(* Logix 5000 project; controller Ceca_1650T_Press 5069-L306ERM rev 32.11; software revision 32.02 *)

TASK MainTask (continuous, watchdog 500 ms) : MainProgram

MODULES
   Local : 5069-L306ERM (5069 0, rev 32.11)
END_MODULES

TYPE Recipe_Setup :
STRUCT
   AUTO_UPPER_ASSIST_POSITION : REAL;
   AUTO_UPPER_LIMIT_POSITION : REAL;
   R_DIECUSHION_AUTO_UP_ASSIST_POSITION : REAL;
   L_DIECUSHION_AUTO_UP_ASSIST_POSITION : REAL;
   L_DIECUSHION_AUTO_UP_LIMIT_POSITION : REAL;
   R_DIECUSHION_AUTO_UP_LIMIT_POSITION : REAL;
   SLIDE_SLOW_DOWN_SIGNAL_POSITION : REAL;
END_STRUCT
END_TYPE

TYPE SICK_AFX60_WS_DATA :   // Data structure for AFS60 / AFM60 WebServer
STRUCT
   Acceleration_Format : INT;
   Acceleration_HighLimit : DINT;
   Acceleration_LowLimit : DINT;
   CMR : DINT;
   CNR_D : DINT;
   CNR_N : DINT;
   CPR : DINT;
   CS : SINT;
   ESF : SINT;
   DirectionChange_Limit : DINT;
   MotionTime_Limit_seconds : DINT;
   PowerTime_Limit_seconds : DINT;
   StartsCCW_Limit : DINT;
   StartsCW_Limit : DINT;
   Position_HighLimit : DINT;
   Position_LowLimit : DINT;
   PresetValue : DINT;
   Scaling : SINT;
   SlaveSignOfLife : DINT;
   Temperature_Format : INT;
   Velocity_Format : INT;
   Velocity_HighLimit : DINT;
   Velocity_LowLimit : DINT;
   xErrorCode : DINT;
   xMsgRecordArray : SINT[4];
   SerialNo : DINT;
END_STRUCT
END_TYPE

ADD_ON_INSTRUCTION SICK_AFX60_A101WS_A103WS_AOI   (* revision 1.0, vendor SICK AG *)
VAR_IN_OUT
   InputAssembly_101WS_103WS : DINT[1]; {required}
   msgGetData : MESSAGE; {required}
   msgSetData : MESSAGE; {required}
   GetData : SICK_AFX60_WS_DATA; {required}
   SetData : SICK_AFX60_WS_DATA; {required}
END_VAR
VAR_INPUT
   ManualGetData : BOOL; {access Read Only}
END_VAR
VAR
   SizeInput : DINT; {access None}
   fbTON : FBD_TIMER; {access None}
   SickAFx_RESET_FaultHeader_Value : SINT; {access None}
   SET_ALL_in_Progress : SINT; {access None}
   Local_ManualGetData : SINT; {access None}
   AttributeList : DINT[24]; {access None}
   Count_Attributes : DINT; {access None}
   ACC_FORMAT : DINT; {access None}
   ACC_HIGH_LIMIT : DINT; {access None}
   ACC_LOW_LIMIT : DINT; {access None}
   CMR : DINT; {access None}
   CNR_D : DINT; {access None}
   CNR_N : DINT; {access None}
   CPR : DINT; {access None}
   CS : DINT; {access None}
   ESF : DINT; {access None}
   MAX_DIR_CHANGE : DINT; {access None}
   MAX_MOTION_TIME : DINT; {access None}
   MAX_POWER_TIME : DINT; {access None}
   MAX_STARTS_CCW : DINT; {access None}
   MAX_STARTS_CW : DINT; {access None}
   POS_HIGH_LIMIT : DINT; {access None}
   POS_LOW_LIMIT : DINT; {access None}
   PRESET_VALUE : DINT; {access None}
   SCALING : DINT; {access None}
   SLAVE_SIGN_OF_LIFE : DINT; {access None}
   TEMP_FORMAT : DINT; {access None}
   VELO_FORMAT : DINT; {access None}
   VELO_HIGH_LIMIT : DINT; {access None}
   VELO_LOW_LIMIT : DINT; {access None}
   arrReadData : DINT[10]; {access None}
   iAttribute : DINT;
   iStep : DINT;
   MAX_ATTRIBUTE : DINT; {access None}
   MIN_ATTRIBUTE : DINT; {access None}
   SERIAL_NO : DINT; {access Read Only}
   goto_iStep : DINT; {access None}
END_VAR

ROUTINE Logic   (* structured text *)
   (*=================================================================================
   Name:	AFX60 WebServer AOI
   Author:	SICK STEGMANN GMBH
   -----------------------------------------------------------------------------------
   Description:
   The routine supports the explicit data messaging between the Rockwell PLC and the
   SICK AFx60 encoder via EtherNet/IP. This routine makes it possible to equalize
   (read and write) a defined set of configuration parameters via EtherNet/IP.
   
   Version history:
   Date        | Version  | created under Logix V. | Author     | Remark
   -----------------------------------------------------------------------------------
   2015.05.21  | 1.0.0    | V21.00.00 CPR 9 SR 5.1 | SICK STD RP| Release version
   2015.06.03  | 1.0.1    | V21.00.00 CPR 9 SR 5.1 | SICK STD RP| AutoSave on Encoder change
   2015.07.06  | 1.0.2    | V21.00.00 CPR 9 SR 5.1 | SICK STD RP| Changed Param Update order
   ==================================================================================*)
   
   (*================================ GENERAL =======================================*)
   (*Initialize variables *)
   	MIN_ATTRIBUTE	:= 0;
   
   	SERIAL_NO      :=  MIN_ATTRIBUTE;
   	ESF            :=  1;
   	SCALING        :=  2;
   	ACC_FORMAT     :=  3;
   	ACC_HIGH_LIMIT :=  4;
   	ACC_LOW_LIMIT  :=  5;
   	CNR_D          :=  6;
   	CNR_N          :=  7;
   	CPR            :=  8;
   	CMR            :=  9;
   	CS             := 10;
   	MAX_DIR_CHANGE := 11;
   	MAX_MOTION_TIME:= 12;
   	MAX_POWER_TIME := 13;
   	MAX_STARTS_CCW := 14;
   	MAX_STARTS_CW  := 15;
   	POS_HIGH_LIMIT := 16;
   	POS_LOW_LIMIT  := 17;
   	PRESET_VALUE   := 18;
   	SLAVE_SIGN_OF_LIFE := 19;
   	TEMP_FORMAT        := 20;
   	VELO_FORMAT        := 21;
   	VELO_HIGH_LIMIT    := 22;
   	VELO_LOW_LIMIT     := 23;
   
   	MAX_ATTRIBUTE 		:= VELO_LOW_LIMIT;
   	Count_Attributes     := MAX_ATTRIBUTE + 1;
   
   	AttributeList[SERIAL_NO      ] :=   6; (* Attrib.ID of SerialNumber - Identity Object *)
   	AttributeList[ACC_FORMAT     ] :=  30; (* Attrib.ID of AccFormat *)
   	AttributeList[ACC_HIGH_LIMIT ] :=  33; (* Attrib.ID of AccHighLimit *)
   	AttributeList[ACC_LOW_LIMIT  ] :=  32; (* Attrib.ID of AccLowLimit *)
   	AttributeList[CMR            ] :=  17; (* Attrib.ID of CMR *)
   	AttributeList[CNR_D          ] := 127; (* Attrib.ID of CNR_D *)
   	AttributeList[CNR_N          ] := 126; (* Attrib.ID of CNR_N *)
   	AttributeList[CPR            ] :=  16; (* Attrib.ID of CPR *)
   	AttributeList[CS             ] :=  12; (* Attrib.ID of CS *)
   	AttributeList[ESF            ] := 125; (* Attrib.ID of ESF *)
   	AttributeList[MAX_DIR_CHANGE ] := 136; (* Attrib.ID of MaxDirChange *)
   	AttributeList[MAX_MOTION_TIME] := 134; (* Attrib.ID of MaxMotionTime *)
   	AttributeList[MAX_POWER_TIME ] := 135; (* Attrib.ID of MaxPowerTime *)
   	AttributeList[MAX_STARTS_CCW ] := 138; (* Attrib.ID of MaxStartsCCW *)
   	AttributeList[MAX_STARTS_CW  ] := 137; (* Attrib.ID of MaxStartsCW *)
   	AttributeList[POS_HIGH_LIMIT ] :=  23; (* Attrib.ID of PosHighLimit *)
   	AttributeList[POS_LOW_LIMIT  ] :=  22; (* Attrib.ID of PosLowLimit *)
   	AttributeList[PRESET_VALUE   ] :=  19; (* Attrib.ID of PresetValue *)
   	AttributeList[SCALING        ] :=  14; (* Attrib.ID of Scaling *)
   	AttributeList[SLAVE_SIGN_OF_LIFE] := 106; (* Attrib.ID of SlaveSignOfLife *)
   	AttributeList[TEMP_FORMAT       ] := 101; (* Attrib.ID of TempFormat *)
   	AttributeList[VELO_FORMAT       ] :=  25; (* Attrib.ID of VeloFormat *)
   	AttributeList[VELO_HIGH_LIMIT   ] :=  28; (* Attrib.ID of VeloHighLimit *)
   	AttributeList[VELO_LOW_LIMIT    ] :=  27; (* Attrib.ID of VeloLowLimit *)
   (* END INIT *)
   
   
   (*================================ GET INPUT DATA =========================*)
   SIZE(InputAssembly_101WS_103WS,0,SizeInput);	(*Size of the input data array*)
   COP(InputAssembly_101WS_103WS[0], arrReadData[0], SizeInput);
   //Assemblies 101WS and 103WS have both Size=3 (DINT-Elements)
   //Assembly   102WS has Size=9 (SINT-Elements)
   
   
   (* manual start reading all parameters (goto step 4) *)
   IF ManualGetData THEN
   	//goto_iStep := 4;
   	iStep := 4;
   	iAttribute := MIN_ATTRIBUTE;
   	SET_ALL_in_Progress := 0;
   END_IF;
   
   
   (*================================ DETECT CHANGES ON WebServer SIDE ==============*)
   (* Step 0: Trigger FaultHeader.Bit15 == 1 *)
   IF arrReadData[0].15 THEN
   	IF iStep=0 THEN
   		// start GET process
   		iStep := 1;
   	END_IF;
   ELSE
   	IF iStep=0 THEN
   		// check if SET process necessary
   		iStep := 8;
   	END_IF;
   END_IF;
   
   
   (*================================ RESET FaultHeader.Bit15 =======================*)
   (* Step 1: Configuration of RESET MSG (RESET Get-Trigger - FaultHeader.Bit15) *)
   IF iStep=1 THEN
   	SickAFx_RESET_FaultHeader_Value := 1; //allways 1
   	msgSetData.REQ_LEN:= 1;
   	COP(SickAFx_RESET_FaultHeader_Value, SetData.xMsgRecordArray[0], msgSetData.REQ_LEN);
   	msgSetData.Class := 35; (* 0x23 PSO *)
   	msgSetData.Instance := 1;
   	msgSetData.Attribute := 139;
   	iStep := 2;
   END_IF;
   
   
   (* Step 2: sending RESET MSG *)
   IF iStep=2 THEN
   	IF NOT msgGetData.EW AND NOT msgGetData.ST AND NOT msgSetData.EW AND NOT msgSetData.ST THEN
   		MSG(msgSetData);
   		fbTON.TimerEnable:= 1;
   		iStep := 3;
   	END_IF;
   END_IF;
   
   
   (* Step 3: msgSetData done, continue reading all get-params *)
   IF iStep=3 AND msgSetData.DN THEN
   	fbTON.TimerEnable:= 0;
   	(* List of GetAttributes finished ? *)
   	IF iAttribute < Count_Attributes THEN
   		(* keep iAttribute unchanged *)
   	ELSE
   		iAttribute := MIN_ATTRIBUTE;
   	END_IF;
   	iStep := 4;
   END_IF;
   
   
   (*================================ GET ALL WebServer Parameters to PLC ===========*)
   (* Step 4: Configuration of GET MSG *)
   IF iStep=4 THEN
   	msgGetData.Class := 35; (* 0x23 PSO *)
   	msgGetData.Instance := 1;
   	msgGetData.Attribute := AttributeList[iAttribute];
   	IF iAttribute=SERIAL_NO THEN
   		msgGetData.Class := 1; 								(* 0x01 Identity Object*)
   		msgGetData.Attribute := AttributeList[SERIAL_NO];
   	END_IF;
   	iStep := 5;
   END_IF;
   
   
   (* Step 5: send GET MSG *)
   IF iStep=5 THEN
   	IF NOT msgGetData.EW AND NOT msgGetData.ST AND NOT msgSetData.EW AND NOT msgSetData.ST THEN
   		MSG(msgGetData);
   		fbTON.TimerEnable:= 1;
   		iStep := 6;
   	END_IF;
   END_IF;
   
   
   IF iStep=6 AND msgGetData.DN THEN
   	fbTON.TimerEnable:= 0;
   	iStep := 7;
   	//Local_ManualGetData := 0;
   	CASE iAttribute OF
   		0: COP(GetData.xMsgRecordArray[0],  GetData.SerialNo, 1);
   			IF SetData.SerialNo <> GetData.SerialNo THEN
   				// NEW Encoder with different SerialNo detected ==> SAVE all PLC params to Encoder
   				SET_ALL_in_Progress := 1;
   				iStep := 8;
   				iAttribute := MIN_ATTRIBUTE;
   				// forcing SET_ALL over manipulated GetData.xxx
   				GetData.Acceleration_Format := SetData.Acceleration_Format + 1 ;
   			 	GetData.Acceleration_HighLimit := SetData.Acceleration_HighLimit + 1 ;
   		 		GetData.Acceleration_LowLimit := SetData.Acceleration_LowLimit + 1 ;
   				GetData.CNR_D := SetData.CNR_D + 1 ;
   				GetData.CNR_N := SetData.CNR_N + 1 ;
   				// Don't set CPR at active ESF: if will be calculated
   				//GetData.CPR := SetData.CPR + 1 ;
   				GetData.CMR := SetData.CMR + 1 ;
   				IF SetData.ESF = 1 THEN
   					//do nothing
   				ELSE
   					GetData.CPR := SetData.CPR + 1 ;
   				END_IF;
   				GetData.CS := SetData.CS + 1 ;
   				GetData.ESF := SetData.ESF + 1 ;
   				GetData.DirectionChange_Limit := SetData.DirectionChange_Limit + 1 ;
   				GetData.MotionTime_Limit_seconds := SetData.MotionTime_Limit_seconds + 1 ;
   				GetData.PowerTime_Limit_seconds := SetData.PowerTime_Limit_seconds + 1 ;
   				GetData.StartsCCW_Limit := SetData.StartsCCW_Limit + 1 ;
   				GetData.StartsCW_Limit  := SetData.StartsCW_Limit + 1 ;
   				GetData.Position_HighLimit := SetData.Position_HighLimit + 1 ;
   				GetData.Position_LowLimit := SetData.Position_LowLimit + 1 ;
   				//GetData.PresetValue := SetData.PresetValue + 1 ; // do NOT SET this param automatically !
   				GetData.Scaling := SetData.Scaling + 1 ;
   				GetData.SlaveSignOfLife := SetData.SlaveSignOfLife + 1 ;
   				GetData.Temperature_Format := SetData.Temperature_Format + 1 ;
   				GetData.Velocity_Format := SetData.Velocity_Format + 1 ;
   				GetData.Velocity_HighLimit := SetData.Velocity_HighLimit + 1 ;
   				GetData.Velocity_LowLimit := SetData.Velocity_LowLimit + 1 ;
   			END_IF;
   			SetData.SerialNo := GetData.SerialNo;
   		1: COP(GetData.xMsgRecordArray[0], GetData.ESF, 1);
   			SetData.ESF := GetData.ESF;
   		2: COP(GetData.xMsgRecordArray[0], GetData.Scaling, 1);
   			SetData.Scaling := GetData.Scaling;
   		3: COP(GetData.xMsgRecordArray[0], GetData.Acceleration_Format, 1);
   			SetData.Acceleration_Format := GetData.Acceleration_Format;
   		4: COP(GetData.xMsgRecordArray[0], GetData.Acceleration_HighLimit, 1);
   			SetData.Acceleration_HighLimit := GetData.Acceleration_HighLimit;
   		5: COP(GetData.xMsgRecordArray[0], GetData.Acceleration_LowLimit, 1);
   			SetData.Acceleration_LowLimit := GetData.Acceleration_LowLimit;
   		6: COP(GetData.xMsgRecordArray[0], GetData.CNR_D, 1);
   			SetData.CNR_D := GetData.CNR_D;
   		7: COP(GetData.xMsgRecordArray[0], GetData.CNR_N, 1);
   			SetData.CNR_N := GetData.CNR_N;
   		8: COP(GetData.xMsgRecordArray[0], GetData.CPR, 1);
   			SetData.CPR := GetData.CPR;
   		9: COP(GetData.xMsgRecordArray[0], GetData.CMR, 1);
   			SetData.CMR := GetData.CMR;
   		10: COP(GetData.xMsgRecordArray[0], GetData.CS, 1);
   			SetData.CS := GetData.CS;
   		11: COP(GetData.xMsgRecordArray[0], GetData.DirectionChange_Limit, 1);
   			SetData.DirectionChange_Limit := GetData.DirectionChange_Limit;
   		12: COP(GetData.xMsgRecordArray[0], GetData.MotionTime_Limit_seconds, 1);
   			SetData.MotionTime_Limit_seconds := GetData.MotionTime_Limit_seconds;
   		13: COP(GetData.xMsgRecordArray[0], GetData.PowerTime_Limit_seconds, 1);
   			SetData.PowerTime_Limit_seconds := GetData.PowerTime_Limit_seconds;
   		14: COP(GetData.xMsgRecordArray[0], GetData.StartsCCW_Limit, 1);
   			SetData.StartsCCW_Limit := GetData.StartsCCW_Limit;
   		15: COP(GetData.xMsgRecordArray[0], GetData.StartsCW_Limit, 1);
   			SetData.StartsCW_Limit := GetData.StartsCW_Limit;
   		16: COP(GetData.xMsgRecordArray[0], GetData.Position_HighLimit, 1);
   			SetData.Position_HighLimit := GetData.Position_HighLimit;
   		17: COP(GetData.xMsgRecordArray[0], GetData.Position_LowLimit, 1);
   			SetData.Position_LowLimit := GetData.Position_LowLimit;
   		18: COP(GetData.xMsgRecordArray[0], GetData.PresetValue, 1);
   			SetData.PresetValue := GetData.PresetValue;
   		19: COP(GetData.xMsgRecordArray[0], GetData.SlaveSignOfLife, 1);
   			SetData.SlaveSignOfLife := GetData.SlaveSignOfLife;
   		20: COP(GetData.xMsgRecordArray[0], GetData.Temperature_Format, 1);
   			SetData.Temperature_Format := GetData.Temperature_Format;
   		21: COP(GetData.xMsgRecordArray[0], GetData.Velocity_Format, 1);
   			SetData.Velocity_Format := GetData.Velocity_Format;
   		22: COP(GetData.xMsgRecordArray[0], GetData.Velocity_HighLimit, 1);
   			SetData.Velocity_HighLimit := GetData.Velocity_HighLimit;
   		23: COP(GetData.xMsgRecordArray[0], GetData.Velocity_LowLimit, 1);
   			SetData.Velocity_LowLimit := GetData.Velocity_LowLimit;
   	END_CASE;
   END_IF;
   
   
   IF iStep=7 THEN
   	iAttribute := iAttribute + 1; (* next attribute index*)
   	IF iAttribute < Count_Attributes THEN
   		iStep := 4; (* continue with next attribute *)
   	ELSE
   		iStep := 8; (* reading all WebServer attributes finished *)
   		iAttribute := MIN_ATTRIBUTE;
   	END_IF;
   END_IF;
   
   
   (*================================ DETECT CHANGES ON PLC Parameters ==============*)
   (* Step 8: check if some changes in PLC tags occured *)
   IF iStep=8 THEN
   	iStep := 0;
   	iAttribute := MIN_ATTRIBUTE;
   	msgSetData.REQ_LEN:= 4; (* other lenghts are defined separately *)
   	IF SetData.SerialNo <> GetData.SerialNo THEN
   		// NEW Encoder with different SerialNo detected ==> SAVE all PLC params to Encoder
   		SET_ALL_in_Progress := 1;
   		iStep := 12;
   		// Forcing SET_ALL over manipulated GetData.xxx
   		GetData.Acceleration_Format := SetData.Acceleration_Format + 2 ;
   	 	GetData.Acceleration_HighLimit := SetData.Acceleration_HighLimit + 2 ;
    		GetData.Acceleration_LowLimit := SetData.Acceleration_LowLimit + 2 ;
   		GetData.CNR_D := SetData.CNR_D + 2 ;
   		GetData.CNR_N := SetData.CNR_N + 2 ;
   		// Don't set CPR at active ESF: if will be calculated
   		//GetData.CPR := SetData.CPR + 2 ;
   		GetData.CMR := SetData.CMR + 2 ;
   		IF SetData.ESF = 1 THEN
   			//do nothing
   		ELSE
   			GetData.CPR := SetData.CPR + 2 ;
   		END_IF;
   		GetData.CS := SetData.CS + 2 ;
   		GetData.ESF := SetData.ESF + 2 ;
   		GetData.DirectionChange_Limit := SetData.DirectionChange_Limit + 2 ;
   		GetData.MotionTime_Limit_seconds := SetData.MotionTime_Limit_seconds + 2 ;
   		GetData.PowerTime_Limit_seconds := SetData.PowerTime_Limit_seconds + 2 ;
   		GetData.StartsCCW_Limit := SetData.StartsCCW_Limit + 2 ;
   		GetData.StartsCW_Limit  := SetData.StartsCW_Limit + 2 ;
   		GetData.Position_HighLimit := SetData.Position_HighLimit + 2 ;
   		GetData.Position_LowLimit := SetData.Position_LowLimit + 2 ;
   		//GetData.PresetValue := SetData.PresetValue + 2 ; // do NOT SET this param automatically !
   		GetData.Scaling := SetData.Scaling + 2 ;
   		GetData.SlaveSignOfLife := SetData.SlaveSignOfLife + 2 ;
   		GetData.Temperature_Format := SetData.Temperature_Format + 2 ;
   		GetData.Velocity_Format := SetData.Velocity_Format + 2 ;
   		GetData.Velocity_HighLimit := SetData.Velocity_HighLimit + 2 ;
   		GetData.Velocity_LowLimit := SetData.Velocity_LowLimit + 2 ;
   		// attribute SerialNo is not settable
   		SetData.SerialNo := GetData.SerialNo;
   	ELSIF SetData.ESF <> GetData.ESF THEN
   		iAttribute := ESF;
   		msgSetData.REQ_LEN := 1;
   		COP(SetData.ESF, SetData.xMsgRecordArray[0], msgSetData.REQ_LEN);
   		iStep := 9;
   	ELSIF SetData.Scaling <> GetData.Scaling THEN
   		iAttribute := SCALING;
   		msgSetData.REQ_LEN := 1;
   		COP(SetData.Scaling, SetData.xMsgRecordArray[0], msgSetData.REQ_LEN);
   		iStep := 9;
   	ELSIF SetData.Acceleration_Format <> GetData.Acceleration_Format THEN
   		iAttribute := ACC_FORMAT;
   		msgSetData.REQ_LEN := 2;
   		COP(SetData.Acceleration_Format, SetData.xMsgRecordArray[0], msgSetData.REQ_LEN);
   		iStep := 9;
   	ELSIF SetData.Acceleration_HighLimit <> GetData.Acceleration_HighLimit THEN
   		iAttribute := ACC_HIGH_LIMIT;
   		COP(SetData.Acceleration_HighLimit, SetData.xMsgRecordArray[0], msgSetData.REQ_LEN);
   		iStep := 9;
   	ELSIF SetData.Acceleration_LowLimit <> GetData.Acceleration_LowLimit THEN
   		iAttribute := ACC_LOW_LIMIT;
   		COP(SetData.Acceleration_LowLimit, SetData.xMsgRecordArray[0], msgSetData.REQ_LEN);
   		iStep := 9;
   	ELSIF SetData.CNR_D <> GetData.CNR_D THEN
   		iAttribute := CNR_D;
   		COP(SetData.CNR_D, SetData.xMsgRecordArray[0], msgSetData.REQ_LEN);
   		iStep := 9;
   	ELSIF SetData.CNR_N <> GetData.CNR_N THEN
   		iAttribute := CNR_N;
   		COP(SetData.CNR_N, SetData.xMsgRecordArray[0], msgSetData.REQ_LEN);
   		iStep := 9;
   	ELSIF SetData.CPR <> GetData.CPR THEN
   		iAttribute := CPR;
   		COP(SetData.CPR, SetData.xMsgRecordArray[0], msgSetData.REQ_LEN);
   		iStep := 9;
   	ELSIF SetData.CMR <> GetData.CMR THEN
   		iAttribute := CMR;
   		COP(SetData.CMR, SetData.xMsgRecordArray[0], msgSetData.REQ_LEN);
   		iStep := 9;
   	ELSIF SetData.CS <> GetData.CS THEN
   		iAttribute := CS;
   		msgSetData.REQ_LEN := 1;
   		COP(SetData.CS, SetData.xMsgRecordArray[0], msgSetData.REQ_LEN);
   		iStep := 9;
   	ELSIF SetData.DirectionChange_Limit <> GetData.DirectionChange_Limit THEN
   		iAttribute := MAX_DIR_CHANGE;
   		COP(SetData.DirectionChange_Limit, SetData.xMsgRecordArray[0], msgSetData.REQ_LEN);
   		iStep := 9;
   	ELSIF SetData.MotionTime_Limit_seconds <> GetData.MotionTime_Limit_seconds THEN
   		iAttribute := MAX_MOTION_TIME;
   		COP(SetData.MotionTime_Limit_seconds, SetData.xMsgRecordArray[0], msgSetData.REQ_LEN);
   		iStep := 9;
   	ELSIF SetData.PowerTime_Limit_seconds <> GetData.PowerTime_Limit_seconds THEN
   		iAttribute := MAX_POWER_TIME;
   		COP(SetData.PowerTime_Limit_seconds, SetData.xMsgRecordArray[0], msgSetData.REQ_LEN);
   		iStep := 9;
   	ELSIF SetData.StartsCCW_Limit <> GetData.StartsCCW_Limit THEN
   		iAttribute := MAX_STARTS_CCW;
   		COP(SetData.StartsCCW_Limit, SetData.xMsgRecordArray[0], msgSetData.REQ_LEN);
   		iStep := 9;
   	ELSIF SetData.StartsCW_Limit <> GetData.StartsCW_Limit THEN
   		iAttribute := MAX_STARTS_CW;
   		COP(SetData.StartsCW_Limit, SetData.xMsgRecordArray[0], msgSetData.REQ_LEN);
   		iStep := 9;
   	ELSIF SetData.Position_HighLimit <> GetData.Position_HighLimit THEN
   		iAttribute := POS_HIGH_LIMIT;
   		COP(SetData.Position_HighLimit, SetData.xMsgRecordArray[0], msgSetData.REQ_LEN);
   		iStep := 9;
   	ELSIF SetData.Position_LowLimit <> GetData.Position_LowLimit THEN
   		iAttribute := POS_LOW_LIMIT;
   		COP(SetData.Position_LowLimit, SetData.xMsgRecordArray[0], msgSetData.REQ_LEN);
   		iStep := 9;
   	ELSIF SetData.PresetValue <> GetData.PresetValue THEN
   		iAttribute := PRESET_VALUE;
   		COP(SetData.PresetValue, SetData.xMsgRecordArray[0], msgSetData.REQ_LEN);
   		iStep := 9;
   	ELSIF SetData.SlaveSignOfLife <> GetData.SlaveSignOfLife THEN
   		iAttribute := SLAVE_SIGN_OF_LIFE;
   		COP(SetData.SlaveSignOfLife, SetData.xMsgRecordArray[0], msgSetData.REQ_LEN);
   		iStep := 9;
   	ELSIF SetData.Temperature_Format <> GetData.Temperature_Format THEN
   		iAttribute := TEMP_FORMAT;
   		msgSetData.REQ_LEN := 2;
   		COP(SetData.Temperature_Format, SetData.xMsgRecordArray[0], msgSetData.REQ_LEN);
   		iStep := 9;
   	ELSIF SetData.Velocity_Format <> GetData.Velocity_Format THEN
   		iAttribute := VELO_FORMAT;
   		msgSetData.REQ_LEN := 2;
   		COP(SetData.Velocity_Format, SetData.xMsgRecordArray[0], msgSetData.REQ_LEN);
   		iStep := 9;
   	ELSIF SetData.Velocity_HighLimit <> GetData.Velocity_HighLimit THEN
   		iAttribute := VELO_HIGH_LIMIT;
   		COP(SetData.Velocity_HighLimit, SetData.xMsgRecordArray[0], msgSetData.REQ_LEN);
   		iStep := 9;
   	ELSIF SetData.Velocity_LowLimit <> GetData.Velocity_LowLimit THEN
   		iAttribute := VELO_LOW_LIMIT;
   		COP(SetData.Velocity_LowLimit, SetData.xMsgRecordArray[0], msgSetData.REQ_LEN);
   		iStep := 9;
   	END_IF;
   END_IF;
   
   
   (*================= SET CHANGED PLC Parameters to the Encoder ====================*)
   (* Step 9: set parameters of actual changed attribute *)
   IF iStep=9 THEN
   	msgSetData.Class := 35; (* 0x23 PSO *)
   	msgSetData.Instance := 1;
   	msgSetData.Attribute := AttributeList[iAttribute];
   	iStep := 10;
   	IF iAttribute = SERIAL_NO THEN
   		iStep := 12;
   	END_IF;
   END_IF;
   
   
   (* Step 10: send SET Mesg. *)
   IF iStep=10 THEN
   	IF NOT msgGetData.EW AND NOT msgGetData.ST AND NOT msgSetData.EW AND NOT msgSetData.ST THEN
   		MSG(msgSetData);
   		fbTON.TimerEnable:= 1;
   		iStep := 11;
   	END_IF;
   END_IF;
   
   
   (* Step 11: assign SetData to GetData *)
   IF iStep=11 AND msgSetData.DN THEN
   	fbTON.TimerEnable:= 0;
   	iStep := 12;
   	CASE iAttribute OF
   		 0: (* do nothing *)
   		 1: GetData.ESF := SetData.ESF;
   		 2: GetData.Scaling := SetData.Scaling;
   		 3: GetData.Acceleration_Format := SetData.Acceleration_Format;
   	 	 4: GetData.Acceleration_HighLimit := SetData.Acceleration_HighLimit;
    		 5: GetData.Acceleration_LowLimit := SetData.Acceleration_LowLimit;
   		 6: GetData.CNR_D := SetData.CNR_D;
   		 7: GetData.CNR_N := SetData.CNR_N;
   		 8: GetData.CPR := SetData.CPR;
   		 9: GetData.CMR := SetData.CMR;
   		10: GetData.CS := SetData.CS;
   		11: GetData.DirectionChange_Limit := SetData.DirectionChange_Limit;
   		12:	GetData.MotionTime_Limit_seconds := SetData.MotionTime_Limit_seconds;
   		13:	GetData.PowerTime_Limit_seconds := SetData.PowerTime_Limit_seconds;
   		14:	GetData.StartsCCW_Limit := SetData.StartsCCW_Limit;
   		15:	GetData.StartsCW_Limit  := SetData.StartsCW_Limit;
   		16: GetData.Position_HighLimit := SetData.Position_HighLimit;
   		17: GetData.Position_LowLimit := SetData.Position_LowLimit;
   		18: GetData.PresetValue := SetData.PresetValue;
   		19: GetData.SlaveSignOfLife := SetData.SlaveSignOfLife;
   		20: GetData.Temperature_Format := SetData.Temperature_Format;
   		21: GetData.Velocity_Format := SetData.Velocity_Format;
   		22: GetData.Velocity_HighLimit := SetData.Velocity_HighLimit;
   		23: GetData.Velocity_LowLimit := SetData.Velocity_LowLimit;
   	END_CASE;
   END_IF;
   
   
   (* Step 12: SET SINGLE / AllInALoop finished *)
   IF iStep=12 THEN
   	IF SET_ALL_in_Progress=1 THEN
   		iStep := 8;
   		IF iAttribute = MAX_ATTRIBUTE THEN
   			SET_ALL_in_Progress := 0;
   			iStep := 4;
   			iAttribute := MIN_ATTRIBUTE;
   		END_IF;
   	ELSE
   		// single SET completed, read all params beginning at step 4.
   		iStep := 4;
   		iAttribute := MIN_ATTRIBUTE;
   	END_IF;
   END_IF;
   
   
   (*================================ DETECT TIMEOUTS ===============================*)
   (*Time out request action*)
   fbTON.PRE:= 10000; //default 10000ms.
   TONR(fbTON);
   IF fbTON.DN THEN
   	(* TIMEOUT reached *)
   	IF iStep=5 THEN
   		GetData.xErrorCode := 16#F001;	(*Error: Read Timeout*)
   	ELSIF iStep=2 OR iStep=10 THEN
   		SetData.xErrorCode := 16#F001;	(*Error: Write Timeout*)
   	END_IF;
   	fbTON.TimerEnable := 0;
   END_IF;
   
   
   (*================================ ERROR INFO ====================================*)
   (* for ErrorCodes see Logix-Help *)
   GetData.xErrorCode := (msgGetData.EXERR*65536) XOR msgGetData.ERR;
   SetData.xErrorCode := (msgSetData.EXERR*65536) XOR msgSetData.ERR;
   
   
   (*================================ DEBUG INFO ====================================*)
   (*GetData.xDebug_iAttrib := iAttribute;
   GetData.xDebug_iStep := iStep;
   GetData.xDebug_SET_ALL_in_Progress := SET_ALL_in_Progress;
   IF ManualGetData THEN
   	GetData.xDebug_ManualGetData := 1;
   ELSE
   	GetData.xDebug_ManualGetData := 0;
   END_IF;
   IF fbTON.TimerEnable THEN
   	GetData.xDebug_TO_TimerEnable := 1;
   ELSE
   	GetData.xDebug_TO_TimerEnable := 0;
   END_IF;
   IF arrReadData[1].7 THEN
   	GetData.xDebug_FH_Bit15 := 1;
   ELSE
   	GetData.xDebug_FH_Bit15 := 0;
   END_IF;*)
   
   // Debug info for STATE MACHINE.
   //iStep := goto_iStep;
   //
   // Use goto_iStep instead of iStep in each case above to set a new step value.
   // See at "IF ManualGetData THEN".
   
   
   (*================================= END =========================================*)
   
   
END_ROUTINE
END_ADD_ON_INSTRUCTION

VAR_GLOBAL   (* controller tags *)
   AIR_PRESSURE_FAULT : BOOL;   // M0029
   AIR_SUPPLY_PRESSURE_DETECT : BOOL;   // B001E
   ANTI_REPEAT : BOOL;   // M0067
   AUTO_CYCLE_ENABLED : BOOL;   // M0014 HMI SELECTION
   AUTO_CYCLE_PREP_COMPLETE : BOOL;   // M0068
   AUTO_CYCLE_SELECTED : BOOL;   // HMI BUTTON/SELECTION B0102
   AUTO_CYCLE_STOP_PB : BOOL;   // B0024
   AUTO_LOWER_LIMIT : BOOL;   // ENCODER SIGNAL B0155
   AUTO_ONE_CYCLE_ENABLED : BOOL;   // M0013 HMI SELECTION
   AUTO_ONE_CYCLE_SELECTED : BOOL;   // HMI BUTTON/SELECTION B0101
   AUTO_RESET_ALLOWED : BOOL;   // M003E
   AUTO_START_PB : BOOL;   // TWO HAND SWITCH DOWN B0022
   AUTO_START_PB_RESET : BOOL;   // TWO HAND SWITCH UP B0023
   AUTO_UPPER_ASSIST : BOOL;   // ENCODER SIGNAL B0152
   AUTO_UPPER_ASSIST_POSITION_MINUS : REAL;
   AUTO_UPPER_ASSIST_POSITION_PLUS : REAL;
   AUTO_UPPER_LIMIT : BOOL;   // ENCODER SIGNAL B0151
   AUTO_UPPER_LIMIT_POSITION_MINUS : REAL;
   AUTO_UPPER_LIMIT_POSITION_PLUS : REAL;
   BLANKING_OFF_SIGNAL : TIMER := (PRE := 150);   // T0018
   BLANKING_PS_ENABLED : BOOL;   // M0018
   BLANKING_PS_SELECT : BOOL;   // B0105 HMI BUTTON
   BOLSTER_CLAMP_OFF_LIMIT : BOOL;   // B0013
   BOLSTER_CLAMP_OFF_VALVE : BOOL;   // B005D
   BOLSTER_CLAMP_ON : BOOL;   // M0006
   BOLSTER_CLAMP_ON_LIMIT : BOOL;   // B0012
   BOLSTER_CLAMP_ON_VALVE : BOOL;   // B005C
   BOLSTER_DISABLED : BOOL;   // M0010
   BOLSTER_ENABLED : BOOL;   // M0011
   BOLSTER_IN_ASSIST_LIMIT : BOOL;   // B000F
   BOLSTER_IN_LIMIT : BOOL;   // B000E
   BOLSTER_IN_PLACE_CLAMPED : BOOL;   // M0037
   BOLSTER_IN_VALVE : BOOL;   // B0059
   BOLSTER_LIFT_PRESSURE_DETECT : BOOL;   // B0019
   BOLSTER_OUT_ASSIST_LIMIT : BOOL;   // B0011
   BOLSTER_OUT_LIMIT : BOOL;   // B0010
   BOLSTER_OUT_VALVE : BOOL;   // B005A
   BOLSTER_REDUCTION_VALVE : BOOL;   // B005B
   BOLSTER_SELECT : BOOL;   // B0108 HMI BUTTON
   BOLSTER_TOUCH_LIMIT_1 : BOOL;   // B0014
   BOLSTER_TOUCH_LIMIT_2 : BOOL;   // B0015
   BOTH_DIE_CUSHIONS_DOWN : BOOL;   // M0036
   BUZZER_SIGNAL : BOOL;   // B0032
   CANCEL_CYLINDER_HIGH_SELECT : BOOL;   // B012F HMI BUTTON
   CANCEL_CYLINDER_LOW_SELECT : BOOL;   // B012E HMI BUTTON
   CANCEL_CYLINDER_LOWER_LIMIT : BOOL;   // B000A
   CANCEL_CYLINDER_UPPER_LIMIT : BOOL;   // B0009
   CANCEL_DECOMPRESSION_VALVE : BOOL;   // B004C
   CANCEL_HIGH_PRESSURE_VAVLE : BOOL;   // B004B
   CANCEL_LOW_PRESSURE_VALVE : BOOL;   // B004A
   CANCEL_UP_VALVE : BOOL;   // B0049
   COOLING_WATER_ON_VALVE : BOOL;   // B0064
   Current_Screen : INT := 4;
   CYCLE_STOP : BOOL;   // M0246
   DC_POWER_ASSIST_VALVE : BOOL;   // B0051
   DEBOUNCE_TIMER_LOCKING_OFF : TIMER := (PRE := 100);   // T0005
   DEBOUNCE_TIMER_LOCKING_OFF_COMPLETE : TIMER := (PRE := 100);   // T0006
   DECOMPRESSION : BOOL;   // M006D
   DIE_CHANGE_ENABLED : BOOL;   // M0015
   DIE_CHANGE_MODE : BOOL;   // HMI BUTTON/SELECTION B0103
   DIE_CLAMPER_CIRCUIT : BOOL;   // K0001
   DIE_CLAMPER_CLAMP_PB : BOOL;   // HMI BUTTON B0118
   DIE_CLAMPER_CLAMPED : BOOL;   // M005B
   DIE_CLAMPER_ON_SELECT : BOOL;   // HMI BUTTON B0117
   DIE_CLAMPER_UNCLAMP_PB : BOOL;   // HMI BUTTON B0119
   DIE_CLAMPER_UNCLAMPED : BOOL;   // M005A
   DIE_CUSHION_1_PAD_SELECT : BOOL;   // B010E HMI BUTTON
   DIE_CUSHION_1_PAD_SELECTED : BOOL;   // M001C
   DIE_CUSHION_2_PAD_L_SELECT : BOOL;   // M001F
   DIE_CUSHION_2_PAD_LEFT_SELECT : BOOL;   // B014E
   DIE_CUSHION_2_PAD_R_SELECT : BOOL;   // M001E
   DIE_CUSHION_2_PAD_RIGHT_SELECT : BOOL;   // B014D
   DIE_CUSHION_2_PAD_SELECT : BOOL;   // B010F HMI BUTTON
   DIE_CUSHION_2_PAD_SELECT_RL : BOOL;   // M001D
   DIE_CUSHION_DOWN_1_PAD : BOOL;   // M004D
   DIE_CUSHION_PB_OFF_STATE : BOOL;   // M003F
   DIE_CUSHION_PUMP_UNLOAD_ASSIST : BOOL;   // M0190
   DIE_CUSHION_UP_1_PAD : BOOL;   // M004C
   DIE_DRAWRIC_CYLINDER_UPPER_PS : BOOL;   // B0018
   DIE_DRAWRIC_DECOMPRESSION_VALVE : BOOL;   // B0056
   DIE_DRAWRIC_DOWN : BOOL;   // M004F
   DIE_DRAWRIC_ON_SELECT : BOOL;   // B0145 HMI BUTTON
   DIE_DRAWRIC_POWER_ASSIST_VALVE : BOOL;   // B0057
   DIE_DRAWRIC_UP : BOOL;   // M004E
   DIE_DRAWRIC_UP_1 : BOOL;   // M007E
   DIE_DRAWRIC_UP_COMPLETE : BOOL;   // M007F
   DIE_DRAWRIC_UP_MEM : TIMER := (PRE := 100);   // T0019
   DIE_SET_CHANGING : BOOL;   // B0037
   DIE_SET_CYLINDER_IN_PB : BOOL;   // B0076
   DIE_SET_CYLINDER_OUT : BOOL;   // M0217
   DIE_SET_CYLINDER_OUT_PB : BOOL;   // B0077
   DIECUSHION_AUTO_START_POSITION : BOOL;   // M0035
   DIECUSHION_PUMP_UNLOADING_VALVE_1 : BOOL;   // B0061
   DIECUSHION_PUMP_UNLOADING_VALVE_2 : BOOL;   // B0063
   DRAW_BLANKING_NOT_SELECT : BOOL;   // M0017
   DRAW_UP_ASSIST : BOOL;   // M007C
   DRAW_UP_ASSIST_COMPLETE : BOOL;   // M007D
   DRAWING_LS_ENABLED : BOOL;   // M0016
   DRAWING_LS_SELECT : BOOL;   // B0104 HMI BUTTON
   EMERGENCY_STOP : BOOL;   // B002A
   ENABLE_1000T : BOOL;   // HMI BUTTON/RECIPE
   ENABLE_1500T : BOOL;   // HMI BUTTON/RECIPE
   ENABLE_500T : BOOL;   // HMI BUTTON/RECIPE
   Fault_Reset_PB : BOOL;
   FILTER_CHOKER : BOOL;   // B001A
   FILTER_CLOGGED_DELAY : TIMER := (PRE := 200);   // T0003
   FILTER_CLOGGED_FAULT : BOOL;   // M0023
   FRONT_SHUTTER_SAFETY : BOOL;   // M002A
   FRONT_SUTTER_ON_LIMIT : BOOL;   // B000C
   HALF_FINISHED_CYLINDER_ADVANCE_LIMIT : BOOL;   // B001B
   HALF_FINISHED_CYLINDER_RETURN_LIMIT : BOOL;   // B001C
   HALF_FINISHED_SUPPLY_VALVE : BOOL;   // B0035
   HMI_START_PUMPS : BOOL;   // HMI BUTTON
   INCH_ENABLED : BOOL;   // M0012 HMI SELECTION
   INCHING_SELECTED : BOOL;   // HMI BUTTON/SELECTION B0100
   Job_Call_Recipe : Recipe_Setup[50];
   L_DIECUSHION_AUTO_UP_ASSIST : BOOL;   // ENCODER SIGNAL B015A
   L_DIECUSHION_AUTO_UP_LIMIT : BOOL;   // B0156 ENCODER SIGNAL
   L_DIECUSHION_CONDITION : BOOL;   // M003B
   L_DIECUSHION_DOWN : BOOL;   // M0003
   L_DIECUSHION_UP : BOOL;   // M0002
   L_DIECUSHION_UP_1 : BOOL;   // M0076
   L_DIECUSHION_UP_ASSIST : BOOL;   // M0074
   L_DIECUSHION_UP_COMPLETE : BOOL;   // M0077
   LEFT_DIECUSHION_DECOMPRESSION_VALVE : BOOL;   // B0054
   LEFT_DIECUSHION_DOWN : BOOL;   // M004B
   LEFT_DIECUSHION_DOWN_PB : BOOL;   // B0113 HMI BUTTON
   LEFT_DIECUSHION_DOWN_VALVE : BOOL;   // B0053
   LEFT_DIECUSHION_LOWER_LIMIT : BOOL;   // B0006
   LEFT_DIECUSHION_POWER_ASSIST_VALVE : BOOL;   // B0055
   LEFT_DIECUSHION_UP : BOOL;   // M004A
   LEFT_DIECUSHION_UP_PB : BOOL;   // B0112 HMI BUTTON
   LEFT_DIECUSHION_UP_VALVE : BOOL;   // B0052
   LEFT_DIECUSHION_UPPER_LIMIT : BOOL;   // B0005
   LEFTDIECUSHIONTIMER : TIMER := (PRE := 1000);
   LIFT_CYLINDER_DOWN_VALVE : BOOL;   // B005F
   LIFT_CYLINDER_UP_VALVE : BOOL;   // B005E
   load_PB : BOOL;
   LOCKING_OFF : BOOL;   // M0004
   LOCKING_OFF_ASSIST : BOOL;   // M0032
   LOCKING_OFF_COMPLETE : BOOL;   // M0033
   LOCKING_OFF_LIMIT : BOOL;   // B0007
   LOCKING_OFF_MEMORY : BOOL;   // M0031
   LOCKING_OFF_VALVE : BOOL;   // B0058
   LOCKING_ON : BOOL;   // M0005
   LOCKING_ON_LIMIT : BOOL;   // B0008
   LUBE_LEVEL_DELAY : TIMER := (PRE := 100);   // T0002
   LUBE_LEVEL_FAULT : BOOL;   // M0022
   LUBRICATION_FAULT : BOOL;   // M0020
   LUBRICATION_OIL_LEVEL_DETECT : BOOL;   // B001F
   LUBRICATION_PRESSURE_DETECT : BOOL;   // B0017
   M_PRESS_AUTO_RUN_COMPLETE : BOOL;   // M0080
   M_PRESS_AUTO_RUN_FINISHED : BOOL;   // M0082
   M_PRESS_AUTO_RUN_FINISHED_TIMER : TIMER := (PRE := 30);   // T0013
   M_PRESS_AUTO_RUN_RESET : BOOL;   // M0083
   M_PRESS_AUTO_RUN_RESET_TIMER : TIMER := (PRE := 30);   // T0014
   M_PRESS_DOWN : BOOL;   // M006A
   M_PRESS_DOWN_COMPLETE : BOOL;   // M006C
   M_PRESS_DOWN_COMPLETE_TIMER : TIMER := (PRE := 30);   // T0012
   M_PRESS_UP : BOOL;   // M006E
   M_PRESS_UP_COMPLETE : BOOL;   // M006F
   Machine_Current_Job : DINT := 4;
   MAIN_DOWN_VALVE : BOOL;   // B0041
   MAIN_DOWN_VALVE_1000_TON : BOOL;   // B0043
   MAIN_DOWN_VALVE_500_TON : BOOL;   // B0042
   MAIN_LOWER_ASSIST_LIMIT : BOOL;   // B0026
   MAIN_LOWER_LIMIT : BOOL;   // B0002
   MAIN_NO_LOAD_VALVE : BOOL;   // B0046
   MAIN_POWER_HOLDING_VALVE : BOOL;   // B0045
   MAIN_PRESS_CONDITION_DOWN : BOOL;   // M0039
   MAIN_PRESS_CONDITION_UP : BOOL;   // M0038
   MAIN_PRESS_DOWN : BOOL;   // M0045
   MAIN_PRESS_DOWN_ASSIST : BOOL;   // M0044
   MAIN_PRESS_NO_PRESSURE_DOWN : BOOL;   // M0047
   MAIN_PRESS_POSITION_SICK : REAL;
   MAIN_PRESS_PRESSURE_DETECT : BOOL;   // B0016
   MAIN_PRESS_SLOW_DOWN : BOOL;   // M0046
   MAIN_PRESS_SLOW_DOWN_SIGNAL : BOOL;   // M0030
   MAIN_PRESS_SLOW_UP : BOOL;   // M0042
   MAIN_PRESS_UP : BOOL;   // M0041
   MAIN_PRESS_UP_ASSIST : BOOL;   // M0040
   MAIN_SLOW_DOWN_VALVE : BOOL;   // B0044
   MAIN_UP_VALVE : BOOL;   // B0040
   MAIN_UPPER_ASSIST : BOOL;   // B0001
   MAIN_UPPER_LIMIT : BOOL;   // B0000
   MOTOR_OVER_LOAD : BOOL;   // B002B
   MOVEMENT_CONFIRMED : BOOL;   // M0064 M0065 M0066
   MOVEMENT_CONFIRMED_TIMER : TIMER := (PRE := 30);   // T0011
   NO_PRESSUE_DOWN_PB : BOOL;   // B010D HMI BUTTON
   OIL_COOLER_START : BOOL;   // B0144
   OIL_TEMP_TOO_HIGH : BOOL;   // B0143
   OIL_TEMP_WARM_UP_ON_SELECT : BOOL;   // B002C HMI BUTTON
   OIL_TEMP_WARM_UP_START : BOOL;   // B0038
   OIL_TEMPERATURE_FAULT : BOOL;   // M0025
   OIL_WORKING_LEVEL_FAULT : BOOL;   // M0021
   ONE_PAD_DIE_CUSHION_UP : BOOL;   // M007A
   ONE_PAD_DIE_CUSHION_UP_ASSIST : BOOL;   // M0078
   ONE_PAD_DIE_CUSHION_UP_COMPLETE : BOOL;   // M007B
   ONE_PAD_DIE_CUSHION_UP_TIMING : TIMER;   // M0079
   OPERATION_ON : BOOL;   // B0020
   PILOT_CHECK_OPEN_VALVE : BOOL;   // B0048
   PILOT_PUMP_HIGH_PRESSURE_VALVE : BOOL;   // B0060
   PILOT_PUMP_MIDDLE_PRESSURE_VALVE : BOOL;   // B0062
   PILOT_PUMP_ON : BOOL;   // B002E
   PREFILL_VALVE_OPEN_VALVE : BOOL;   // B0047
   PREFILL_VALVE_OPEN_VALVE_2 : BOOL;   // B0066
   PRESS_AUTO_CYCLE_SELECT_CONDITION : BOOL;   // M0060
   PRESS_AUTO_RUN : BOOL;   // M0069
   PRESS_AUTO_START_POSITION : BOOL;   // M0063
   PRESS_AUTO_START_POSITION_ASSIST : BOOL;   // M0062
   PRESS_HAS_A_FAULT : BOOL;   // M0027
   PRESS_HAS_A_FAULT_2 : BOOL;   // M0028
   PRESS_HOLDING_TIME : BOOL;   // M006B
   PRESS_HOLDING_TIMER : TIMER := (PRE := 1000);   // PRESS HOLDING TIMER
   PRESS_READY_CONFIRM : BOOL;   // M0043
   PUMP_ON_DELAY_CHECK : TIMER := (PRE := 300);   // T0000
   PUMP_RUN : BOOL;   // B0021
   PUMP_START : BOOL;   // B1000
   PUMP_STOP_SIGNAL : BOOL;   // B0030
   R_DIECUSHION_AUTO_UP_ASSIST : BOOL;   // B015B ENCODER SIGNAL
   R_DIECUSHION_AUTO_UP_LIMIT : BOOL;   // B0158 ENCODER SIGNAL
   R_DIECUSHION_DOWN : BOOL;   // M0001
   R_DIECUSHION_UP : BOOL;   // M0000
   R_DIECUSHION_UP_1 : BOOL;   // M0072
   R_DIECUSHION_UP_ASSIST : BOOL;   // M0070
   R_DIECUSHION_UP_COMPLETE : BOOL;   // M0073
   REAR_SHUTTER_ON_LIMIT : BOOL;   // B000D
   Recipe_Max : DINT := 40;
   Recipe_Name_Pointer : DINT := 4;
   Recipe_Number : COUNTER := (PRE := 11, ACC := 4);
   RESET_PB : BOOL;   // HMI RESET PB
   RESETTING_CONFIRMATION : BOOL;   // M0061
   RIGHT_DIECUSHION_CONDITION : BOOL;   // M003A
   RIGHT_DIECUSHION_DECOMPRESSION_VALVE : BOOL;   // B004F
   RIGHT_DIECUSHION_DOWN : BOOL;   // M0049
   RIGHT_DIECUSHION_DOWN_PB : BOOL;   // B0111 HMI BUTTON
   RIGHT_DIECUSHION_DOWN_VALVE : BOOL;   // B004E
   RIGHT_DIECUSHION_LOWER_LIMIT : BOOL;   // B0004
   RIGHT_DIECUSHION_POWER_ASSIST_VALVE : BOOL;   // B0050
   RIGHT_DIECUSHION_UP : BOOL;   // M0048
   RIGHT_DIECUSHION_UP_PB : BOOL;   // B0110 HMI BUTTON
   RIGHT_DIECUSHION_UP_VALVE : BOOL;   // B004D
   RIGHT_DIECUSHION_UPPER_LIMIT : BOOL;   // B0003
   RIGHTDIECUSHIONTIMER : TIMER := (PRE := 1000);
   SAFETY_BAR_OPENED : BOOL;   // B000B
   Save_Delay : TIMER;
   save_pb : BOOL;
   Screen_Control : INT;
   Scroll_Down : BOOL;
   Scroll_up : BOOL;
   SickAFxWS_Enc1_AOI : SICK_AFX60_A101WS_A103WS_AOI;
   SickAFxWS_Enc1_Cyclic_GetSet : BOOL := 1;
   SickAFxWS_Enc1_GetData : SICK_AFX60_WS_DATA := (Acceleration_Format := 2064, Acceleration_HighLimit := 1073741823, Acceleration_LowLimit := -1073741823, CMR := 6144000, CNR_D := 1, CNR_N := 2048, CPR := 1500, DirectionChange_Limit := 1000000, MotionTime_Limit_seconds := 630720000, PowerTime_Limit_seconds := 630720000, StartsCCW_Limit := 1000000, StartsCW_Limit := 1000000, Position_HighLimit := 6143999, Scaling := 1, SlaveSignOfLife := 1281, Temperature_Format := 4609, Velocity_Format := 7951, Velocity_HighLimit := 150, Velocity_LowLimit := -150, xMsgRecordArray[0] := 106, xMsgRecordArray[1] := -1, xMsgRecordArray[2] := -1, xMsgRecordArray[3] := -1, SerialNo := 285868907);
   SickAFxWS_Enc1_Init_GetSet : BOOL;
   SickAFxWS_Enc1_msgGetData : MESSAGE;
        MessageParameters(ServiceCode := 16#000e, DestinationTag := SickAFxWS_Enc1_GetData.xMsgRecordArray[0], ...)
   SickAFxWS_Enc1_msgSetData : MESSAGE;
        MessageParameters(ServiceCode := 16#0010, LocalElement := SickAFxWS_Enc1_SetData.xMsgRecordArray[0], ...)
   SickAFxWS_Enc1_SetData : SICK_AFX60_WS_DATA := (Acceleration_Format := 2064, Acceleration_HighLimit := 1073741823, Acceleration_LowLimit := -1073741823, CMR := 6144000, CNR_D := 1, CNR_N := 2048, CPR := 1500, DirectionChange_Limit := 1000000, MotionTime_Limit_seconds := 630720000, PowerTime_Limit_seconds := 630720000, StartsCCW_Limit := 1000000, StartsCW_Limit := 1000000, Position_HighLimit := 6143999, Scaling := 1, SlaveSignOfLife := 1281, Temperature_Format := 4609, Velocity_Format := 7951, Velocity_HighLimit := 150, Velocity_LowLimit := -150, xMsgRecordArray[0] := 1, xMsgRecordArray[1] := 18, xMsgRecordArray[2] := -1, xMsgRecordArray[3] := -1, SerialNo := 285868907);
        .Temperature_Format   // 4608 = Celsius 4609 =Fahrenheit
        .Scaling   // 0= Scaling Disabled 1= Scaling Enabled
        .SlaveSignOfLife   // 1280=Heartbeat Off 1281=Hearbeat ON
   SickAFxWS_Enc1_Timer_GetSet : TIMER := (PRE := 100, ACC := 47, EN := 1, TT := 1);
   SLIDE_DOWN_PB : BOOL;   // B010B HMI BUTTON
   SLIDE_SLOW_DOWN_PB : BOOL;   // B010C HMI BUTTON
   SLIDE_SLOW_DOWN_SIGNAL : BOOL;   // B0154 ENCODER SIGNAL
   SLIDE_SLOW_DOWN_SIGNAL_POSITION_MINUS : REAL;
   SLIDE_SLOW_DOWN_SIGNAL_POSITION_PLUS : REAL;
   SLIDE_SLOW_UP_PB : BOOL;   // B010A HMI BUTTON
   SLIDE_UP_PB : BOOL;   // HMI BUTTON B0109
   TIMER_OFF_DELAY_1500T : TIMER := (PRE := 50);   // T0017
   TIMER_OFF_DELAY_500T : TIMER := (PRE := 10);   // T0016
   TRM1 : BOOL;   // B1003
   TRM1_TIMER : TIMER := (PRE := 5000);   // 5 SECONDS
   TRM2 : BOOL;   // B1001
   TRM2_TIMER : TIMER := (PRE := 5000);   // 5 SECONDS
   TRM3 : BOOL;   // B1002
   TRM3_TIMER : TIMER := (PRE := 1000);   // 1 SECOND
   UPPER_DIE_CLAMP_ON_DETECT : BOOL;   // B001D
   UPPER_DIECLAMP_OFF_VALVE : BOOL;   // B0065
   WARM_UP_FINISHED : BOOL;   // M009E
   WARM_UP_OFF_TEMP : BOOL;   // B0027
   WARM_UP_ON : BOOL;   // M009D
   WARM_UP_ON_TIMING : TIMER := (PRE := 200);   // T0023
   WARM_UP_SELECT_OFF_TIMER : TIMER := (PRE := 100);   // T0024
   WARM_UP_SELECT_ON_TIMER : TIMER := (PRE := 100);   // T0025
   WORK_LOCATION_VALVE : BOOL;   // B0036
   WORKING_LEVEL_DELAY_CHECK : TIMER := (PRE := 100);   // T0001
   WORKING_OIL_LEVEL_DETECT : BOOL;   // B0025
END_VAR

PROGRAM MainProgram   (* main routine MainRoutine *)
VAR
   STATUS_MESSAGE : STRING;
END_VAR

ROUTINE Auto_Cycle   (* ladder *)
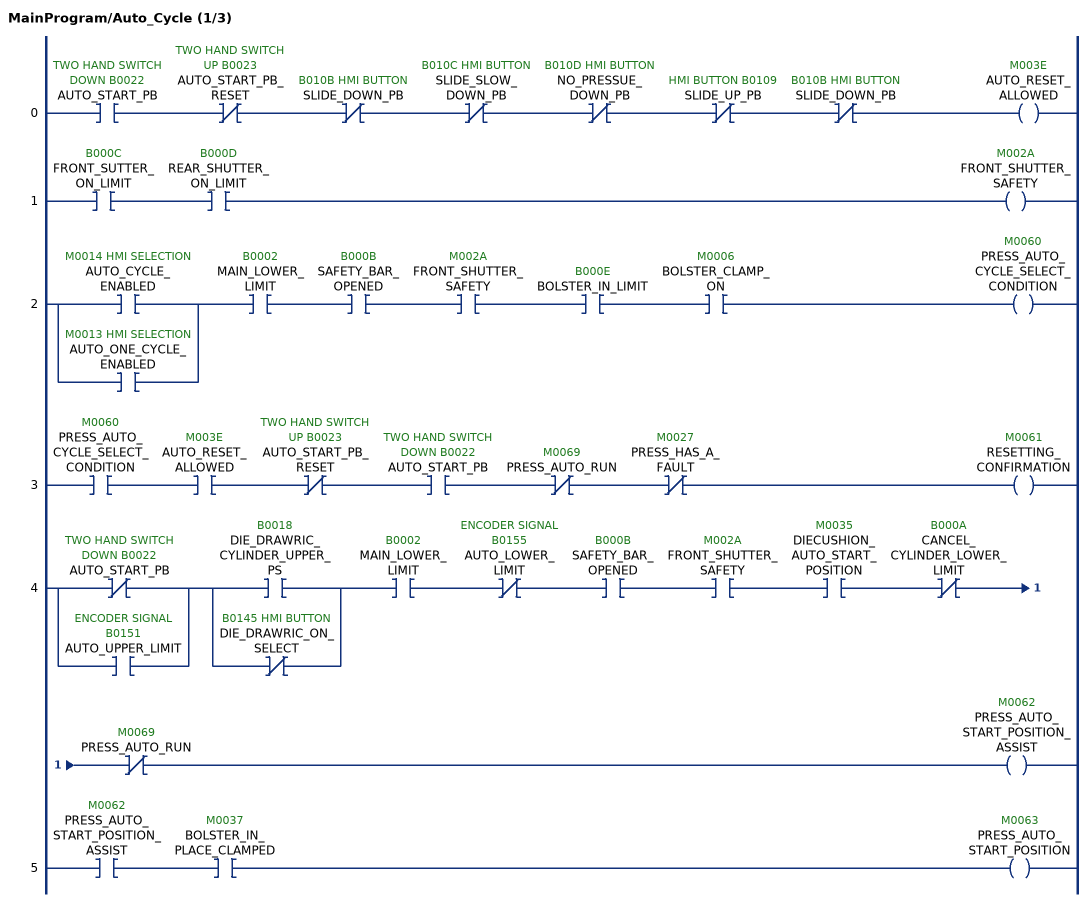
   0: XIC(AUTO_START_PB)XIO(AUTO_START_PB_RESET)XIO(SLIDE_DOWN_PB)XIO(SLIDE_SLOW_DOWN_PB)XIO(NO_PRESSUE_DOWN_PB)XIO(SLIDE_UP_PB)XIO(SLIDE_DOWN_PB)OTE(AUTO_RESET_ALLOWED);
   1: XIC(FRONT_SUTTER_ON_LIMIT)XIC(REAR_SHUTTER_ON_LIMIT)OTE(FRONT_SHUTTER_SAFETY);
   2: [XIC(AUTO_CYCLE_ENABLED) ,XIC(AUTO_ONE_CYCLE_ENABLED) ]XIC(MAIN_LOWER_LIMIT)XIC(SAFETY_BAR_OPENED)XIC(FRONT_SHUTTER_SAFETY)XIC(BOLSTER_IN_LIMIT)XIC(BOLSTER_CLAMP_ON)OTE(PRESS_AUTO_CYCLE_SELECT_CONDITION);
   3: XIC(PRESS_AUTO_CYCLE_SELECT_CONDITION)XIC(AUTO_RESET_ALLOWED)XIO(AUTO_START_PB_RESET)XIC(AUTO_START_PB)XIO(PRESS_AUTO_RUN)XIO(PRESS_HAS_A_FAULT)OTE(RESETTING_CONFIRMATION);
   4: [XIO(AUTO_START_PB) ,XIC(AUTO_UPPER_LIMIT) ][XIC(DIE_DRAWRIC_CYLINDER_UPPER_PS) ,XIO(DIE_DRAWRIC_ON_SELECT) ]XIC(MAIN_LOWER_LIMIT)XIO(AUTO_LOWER_LIMIT)XIC(SAFETY_BAR_OPENED)XIC(FRONT_SHUTTER_SAFETY)XIC(DIECUSHION_AUTO_START_POSITION)XIO(CANCEL_CYLINDER_LOWER_LIMIT)XIO(PRESS_AUTO_RUN)OTE(PRESS_AUTO_START_POSITION_ASSIST);
   5: XIC(PRESS_AUTO_START_POSITION_ASSIST)XIC(BOLSTER_IN_PLACE_CLAMPED)OTE(PRESS_AUTO_START_POSITION);
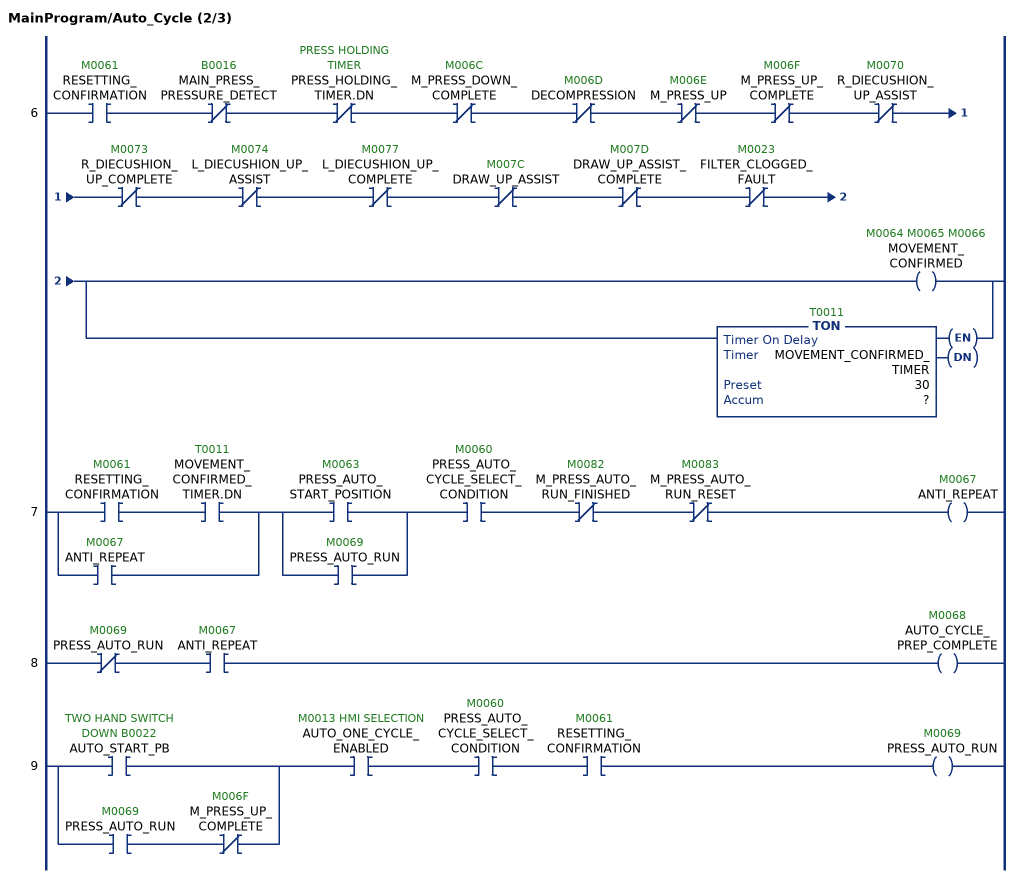
   6: XIC(RESETTING_CONFIRMATION)XIO(MAIN_PRESS_PRESSURE_DETECT)XIO(PRESS_HOLDING_TIMER.DN)XIO(M_PRESS_DOWN_COMPLETE)XIO(DECOMPRESSION)XIO(M_PRESS_UP)XIO(M_PRESS_UP_COMPLETE)XIO(R_DIECUSHION_UP_ASSIST)XIO(R_DIECUSHION_UP_COMPLETE)XIO(L_DIECUSHION_UP_ASSIST)XIO(L_DIECUSHION_UP_COMPLETE)XIO(DRAW_UP_ASSIST)XIO(DRAW_UP_ASSIST_COMPLETE)XIO(FILTER_CLOGGED_FAULT)[OTE(MOVEMENT_CONFIRMED) ,TON(MOVEMENT_CONFIRMED_TIMER,?,?) ];
   7: [XIC(RESETTING_CONFIRMATION) XIC(MOVEMENT_CONFIRMED_TIMER.DN) ,XIC(ANTI_REPEAT) ][XIC(PRESS_AUTO_START_POSITION) ,XIC(PRESS_AUTO_RUN) ]XIC(PRESS_AUTO_CYCLE_SELECT_CONDITION)XIO(M_PRESS_AUTO_RUN_FINISHED)XIO(M_PRESS_AUTO_RUN_RESET)OTE(ANTI_REPEAT);
   8: XIO(PRESS_AUTO_RUN)XIC(ANTI_REPEAT)OTE(AUTO_CYCLE_PREP_COMPLETE);
   9: [XIC(AUTO_START_PB) ,XIC(PRESS_AUTO_RUN) XIO(M_PRESS_UP_COMPLETE) ]XIC(AUTO_ONE_CYCLE_ENABLED)XIC(PRESS_AUTO_CYCLE_SELECT_CONDITION)XIC(RESETTING_CONFIRMATION)OTE(PRESS_AUTO_RUN);
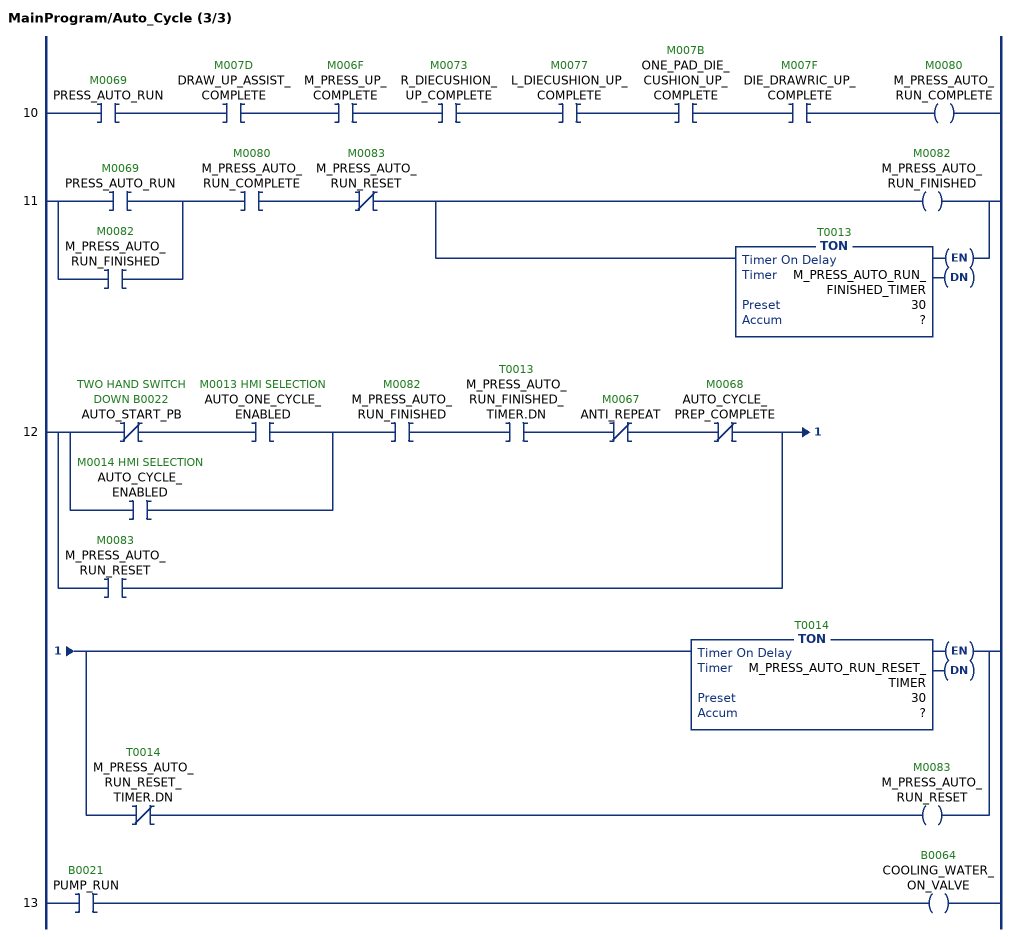
   10: XIC(PRESS_AUTO_RUN)XIC(DRAW_UP_ASSIST_COMPLETE)XIC(M_PRESS_UP_COMPLETE)XIC(R_DIECUSHION_UP_COMPLETE)XIC(L_DIECUSHION_UP_COMPLETE)XIC(ONE_PAD_DIE_CUSHION_UP_COMPLETE)XIC(DIE_DRAWRIC_UP_COMPLETE)OTE(M_PRESS_AUTO_RUN_COMPLETE);
   11: [XIC(PRESS_AUTO_RUN) ,XIC(M_PRESS_AUTO_RUN_FINISHED) ]XIC(M_PRESS_AUTO_RUN_COMPLETE)XIO(M_PRESS_AUTO_RUN_RESET)[OTE(M_PRESS_AUTO_RUN_FINISHED) ,TON(M_PRESS_AUTO_RUN_FINISHED_TIMER,?,?) ];
   12: [[XIO(AUTO_START_PB) XIC(AUTO_ONE_CYCLE_ENABLED) ,XIC(AUTO_CYCLE_ENABLED) ] XIC(M_PRESS_AUTO_RUN_FINISHED) XIC(M_PRESS_AUTO_RUN_FINISHED_TIMER.DN) XIO(ANTI_REPEAT) XIO(AUTO_CYCLE_PREP_COMPLETE) ,XIC(M_PRESS_AUTO_RUN_RESET) ][TON(M_PRESS_AUTO_RUN_RESET_TIMER,?,?) ,XIO(M_PRESS_AUTO_RUN_RESET_TIMER.DN) OTE(M_PRESS_AUTO_RUN_RESET) ];
   13: XIC(PUMP_RUN)OTE(COOLING_WATER_ON_VALVE);
END_ROUTINE

ROUTINE Blanking   (* ladder *)
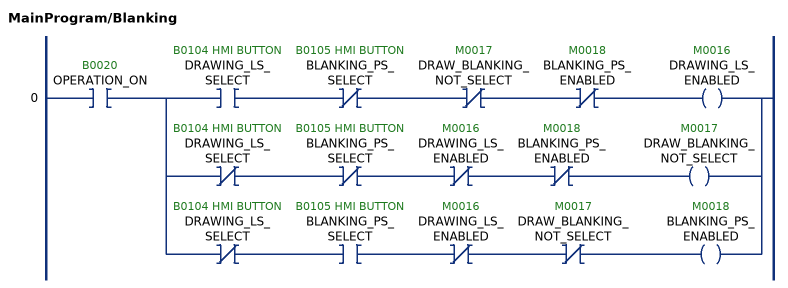
   0: XIC(OPERATION_ON)[XIC(DRAWING_LS_SELECT) XIO(BLANKING_PS_SELECT) XIO(DRAW_BLANKING_NOT_SELECT) XIO(BLANKING_PS_ENABLED) OTE(DRAWING_LS_ENABLED) ,XIO(DRAWING_LS_SELECT) XIO(BLANKING_PS_SELECT) XIO(DRAWING_LS_ENABLED) XIO(BLANKING_PS_ENABLED) OTE(DRAW_BLANKING_NOT_SELECT) ,XIO(DRAWING_LS_SELECT) XIC(BLANKING_PS_SELECT) XIO(DRAWING_LS_ENABLED) XIO(DRAW_BLANKING_NOT_SELECT) OTE(BLANKING_PS_ENABLED) ];
END_ROUTINE

ROUTINE Bolster   (* ladder *)
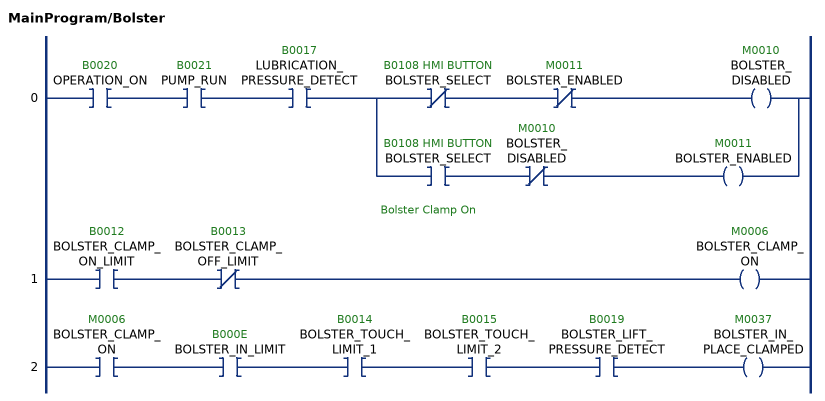
   0: XIC(OPERATION_ON)XIC(PUMP_RUN)XIC(LUBRICATION_PRESSURE_DETECT)[XIO(BOLSTER_SELECT) XIO(BOLSTER_ENABLED) OTE(BOLSTER_DISABLED) ,XIC(BOLSTER_SELECT) XIO(BOLSTER_DISABLED) OTE(BOLSTER_ENABLED) ];
   // Bolster Clamp On
   1: XIC(BOLSTER_CLAMP_ON_LIMIT)XIO(BOLSTER_CLAMP_OFF_LIMIT)OTE(BOLSTER_CLAMP_ON);
   2: XIC(BOLSTER_CLAMP_ON)XIC(BOLSTER_IN_LIMIT)XIC(BOLSTER_TOUCH_LIMIT_1)XIC(BOLSTER_TOUCH_LIMIT_2)XIC(BOLSTER_LIFT_PRESSURE_DETECT)OTE(BOLSTER_IN_PLACE_CLAMPED);
END_ROUTINE

ROUTINE Cancel_Valves   (* ladder *)
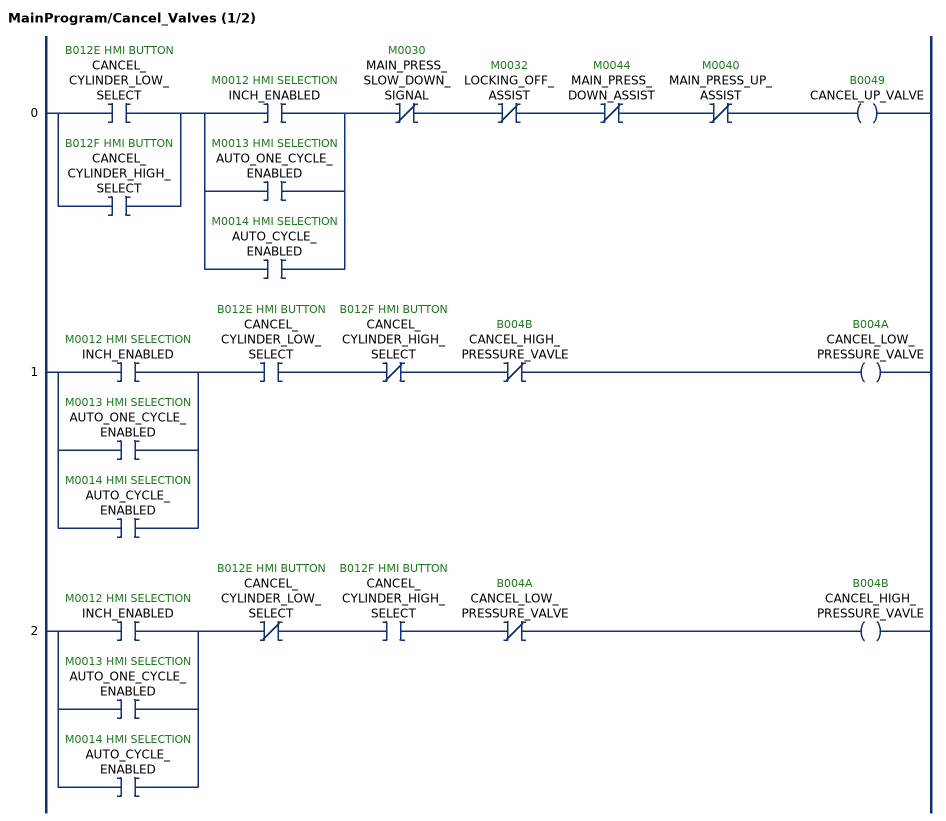
   0: [XIC(CANCEL_CYLINDER_LOW_SELECT) ,XIC(CANCEL_CYLINDER_HIGH_SELECT) ][XIC(INCH_ENABLED) ,XIC(AUTO_ONE_CYCLE_ENABLED) ,XIC(AUTO_CYCLE_ENABLED) ]XIO(MAIN_PRESS_SLOW_DOWN_SIGNAL)XIO(LOCKING_OFF_ASSIST)XIO(MAIN_PRESS_DOWN_ASSIST)XIO(MAIN_PRESS_UP_ASSIST)OTE(CANCEL_UP_VALVE);
   1: [XIC(INCH_ENABLED) ,XIC(AUTO_ONE_CYCLE_ENABLED) ,XIC(AUTO_CYCLE_ENABLED) ]XIC(CANCEL_CYLINDER_LOW_SELECT)XIO(CANCEL_CYLINDER_HIGH_SELECT)XIO(CANCEL_HIGH_PRESSURE_VAVLE)OTE(CANCEL_LOW_PRESSURE_VALVE);
   2: [XIC(INCH_ENABLED) ,XIC(AUTO_ONE_CYCLE_ENABLED) ,XIC(AUTO_CYCLE_ENABLED) ]XIO(CANCEL_CYLINDER_LOW_SELECT)XIC(CANCEL_CYLINDER_HIGH_SELECT)XIO(CANCEL_LOW_PRESSURE_VALVE)OTE(CANCEL_HIGH_PRESSURE_VAVLE);
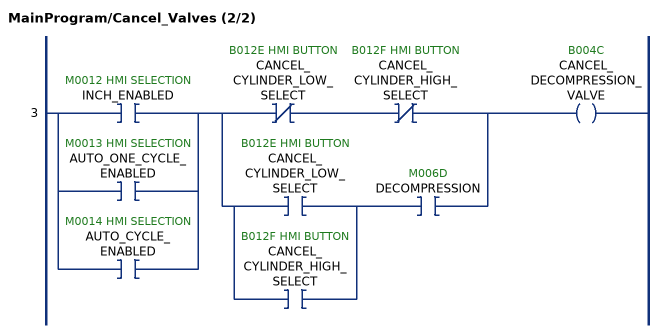
   3: [XIC(INCH_ENABLED) ,XIC(AUTO_ONE_CYCLE_ENABLED) ,XIC(AUTO_CYCLE_ENABLED) ][XIO(CANCEL_CYLINDER_LOW_SELECT) XIO(CANCEL_CYLINDER_HIGH_SELECT) ,[XIC(CANCEL_CYLINDER_LOW_SELECT) ,XIC(CANCEL_CYLINDER_HIGH_SELECT) ] XIC(DECOMPRESSION) ]OTE(CANCEL_DECOMPRESSION_VALVE);
END_ROUTINE

ROUTINE Die_Clamp   (* ladder *)
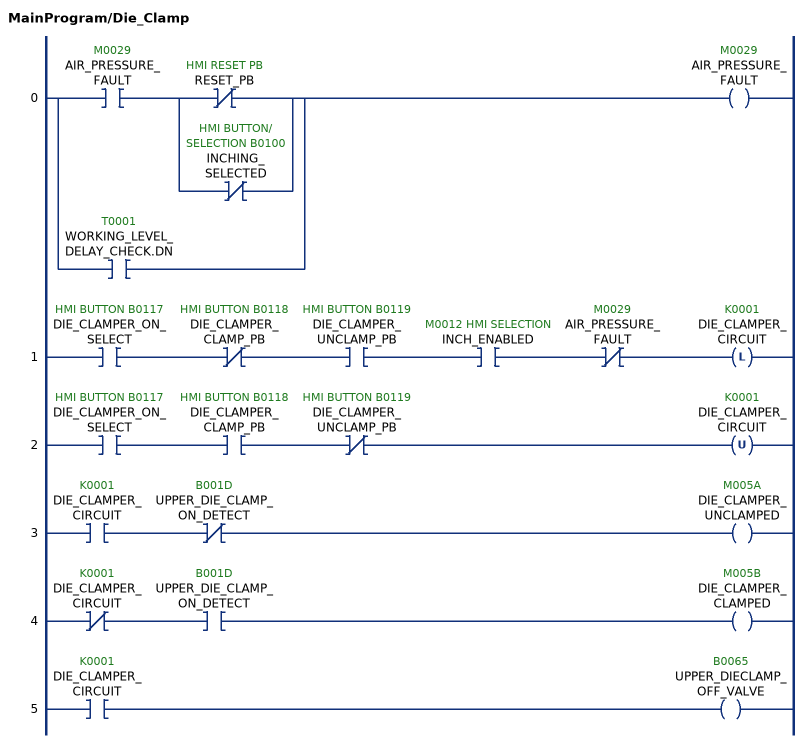
   0: [XIC(AIR_PRESSURE_FAULT) [XIO(RESET_PB) ,XIO(INCHING_SELECTED) ] ,XIC(WORKING_LEVEL_DELAY_CHECK.DN) ]OTE(AIR_PRESSURE_FAULT);
   1: XIC(DIE_CLAMPER_ON_SELECT)XIO(DIE_CLAMPER_CLAMP_PB)XIC(DIE_CLAMPER_UNCLAMP_PB)XIC(INCH_ENABLED)XIO(AIR_PRESSURE_FAULT)OTL(DIE_CLAMPER_CIRCUIT);
   2: XIC(DIE_CLAMPER_ON_SELECT)XIC(DIE_CLAMPER_CLAMP_PB)XIO(DIE_CLAMPER_UNCLAMP_PB)OTU(DIE_CLAMPER_CIRCUIT);
   3: XIC(DIE_CLAMPER_CIRCUIT)XIO(UPPER_DIE_CLAMP_ON_DETECT)OTE(DIE_CLAMPER_UNCLAMPED);
   4: XIO(DIE_CLAMPER_CIRCUIT)XIC(UPPER_DIE_CLAMP_ON_DETECT)OTE(DIE_CLAMPER_CLAMPED);
   5: XIC(DIE_CLAMPER_CIRCUIT)OTE(UPPER_DIECLAMP_OFF_VALVE);
END_ROUTINE

ROUTINE Die_Cushion   (* ladder *)
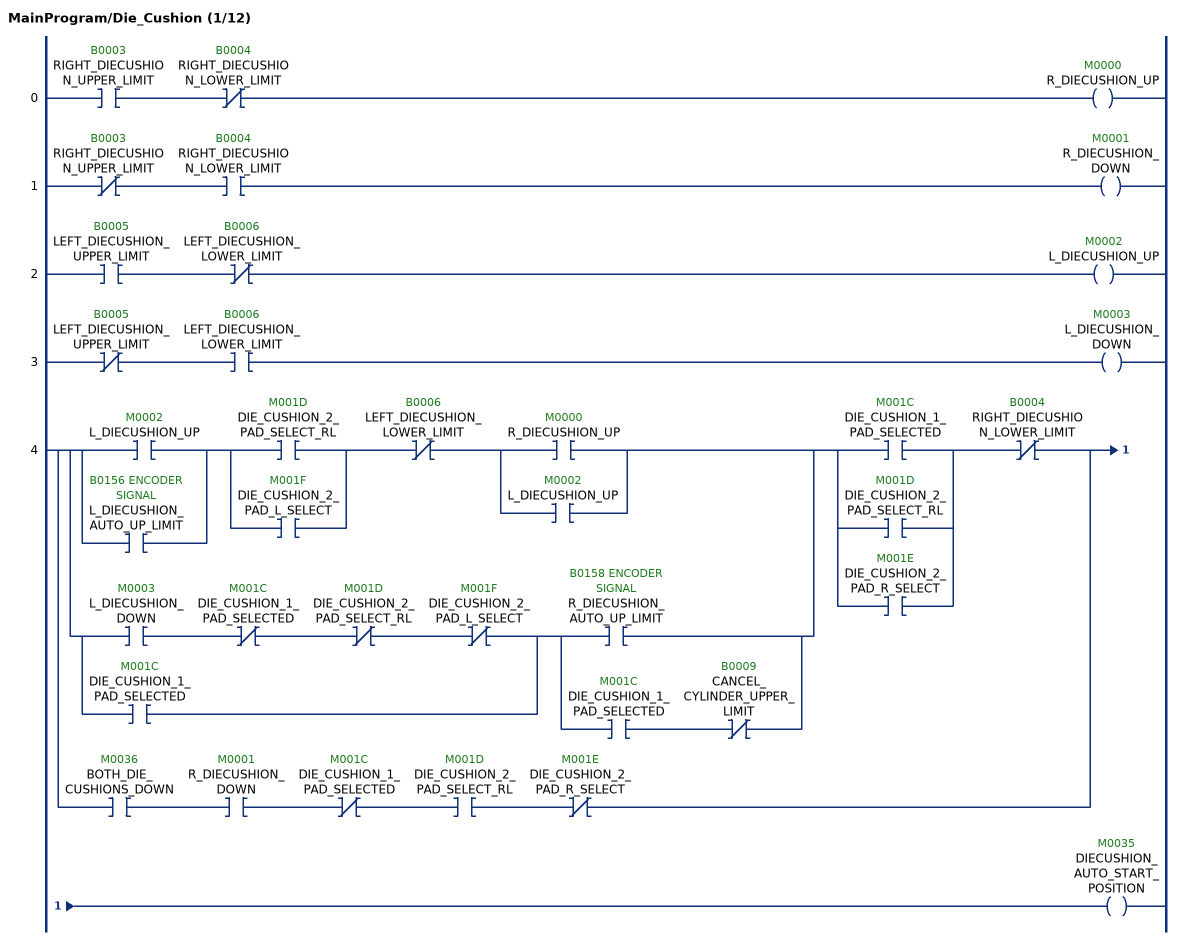
   0: XIC(RIGHT_DIECUSHION_UPPER_LIMIT)XIO(RIGHT_DIECUSHION_LOWER_LIMIT)OTE(R_DIECUSHION_UP);
   1: XIO(RIGHT_DIECUSHION_UPPER_LIMIT)XIC(RIGHT_DIECUSHION_LOWER_LIMIT)OTE(R_DIECUSHION_DOWN);
   2: XIC(LEFT_DIECUSHION_UPPER_LIMIT)XIO(LEFT_DIECUSHION_LOWER_LIMIT)OTE(L_DIECUSHION_UP);
   3: XIO(LEFT_DIECUSHION_UPPER_LIMIT)XIC(LEFT_DIECUSHION_LOWER_LIMIT)OTE(L_DIECUSHION_DOWN);
   4: [[[XIC(L_DIECUSHION_UP) ,XIC(L_DIECUSHION_AUTO_UP_LIMIT) ] [XIC(DIE_CUSHION_2_PAD_SELECT_RL) ,XIC(DIE_CUSHION_2_PAD_L_SELECT) ] XIO(LEFT_DIECUSHION_LOWER_LIMIT) [XIC(R_DIECUSHION_UP) ,XIC(L_DIECUSHION_UP) ] ,[XIC(L_DIECUSHION_DOWN) XIO(DIE_CUSHION_1_PAD_SELECTED) XIO(DIE_CUSHION_2_PAD_SELECT_RL) XIO(DIE_CUSHION_2_PAD_L_SELECT) ,XIC(DIE_CUSHION_1_PAD_SELECTED) ] [XIC(R_DIECUSHION_AUTO_UP_LIMIT) ,XIC(DIE_CUSHION_1_PAD_SELECTED) XIO(CANCEL_CYLINDER_UPPER_LIMIT) ] ] [XIC(DIE_CUSHION_1_PAD_SELECTED) ,XIC(DIE_CUSHION_2_PAD_SELECT_RL) ,XIC(DIE_CUSHION_2_PAD_R_SELECT) ] XIO(RIGHT_DIECUSHION_LOWER_LIMIT) ,XIC(BOTH_DIE_CUSHIONS_DOWN) XIC(R_DIECUSHION_DOWN) XIO(DIE_CUSHION_1_PAD_SELECTED) XIC(DIE_CUSHION_2_PAD_SELECT_RL) XIO(DIE_CUSHION_2_PAD_R_SELECT) ]OTE(DIECUSHION_AUTO_START_POSITION);
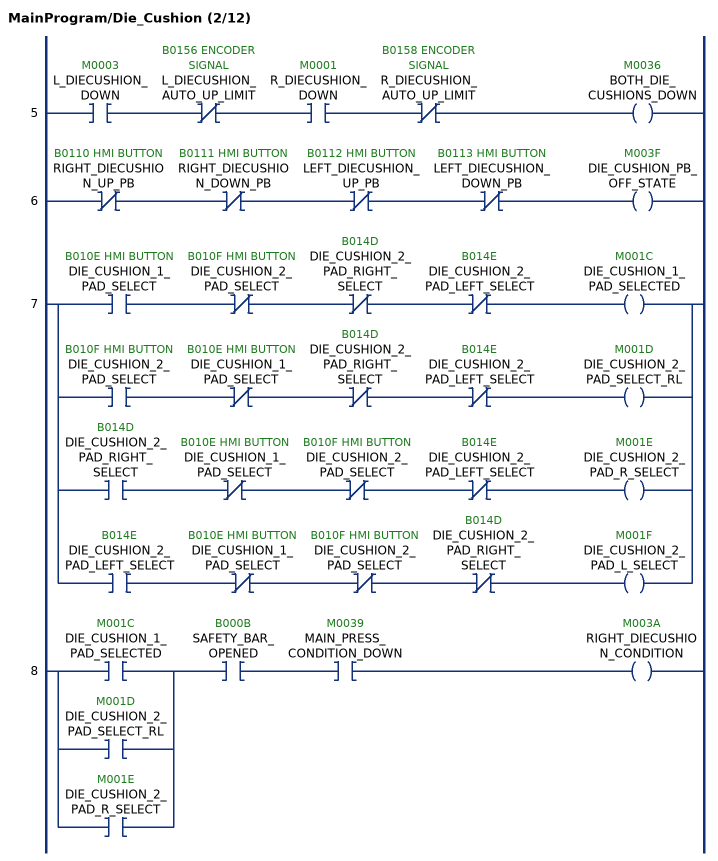
   5: XIC(L_DIECUSHION_DOWN)XIO(L_DIECUSHION_AUTO_UP_LIMIT)XIC(R_DIECUSHION_DOWN)XIO(R_DIECUSHION_AUTO_UP_LIMIT)OTE(BOTH_DIE_CUSHIONS_DOWN);
   6: XIO(RIGHT_DIECUSHION_UP_PB)XIO(RIGHT_DIECUSHION_DOWN_PB)XIO(LEFT_DIECUSHION_UP_PB)XIO(LEFT_DIECUSHION_DOWN_PB)OTE(DIE_CUSHION_PB_OFF_STATE);
   7: [XIC(DIE_CUSHION_1_PAD_SELECT) XIO(DIE_CUSHION_2_PAD_SELECT) XIO(DIE_CUSHION_2_PAD_RIGHT_SELECT) XIO(DIE_CUSHION_2_PAD_LEFT_SELECT) OTE(DIE_CUSHION_1_PAD_SELECTED) ,XIC(DIE_CUSHION_2_PAD_SELECT) XIO(DIE_CUSHION_1_PAD_SELECT) XIO(DIE_CUSHION_2_PAD_RIGHT_SELECT) XIO(DIE_CUSHION_2_PAD_LEFT_SELECT) OTE(DIE_CUSHION_2_PAD_SELECT_RL) ,XIC(DIE_CUSHION_2_PAD_RIGHT_SELECT) XIO(DIE_CUSHION_1_PAD_SELECT) XIO(DIE_CUSHION_2_PAD_SELECT) XIO(DIE_CUSHION_2_PAD_LEFT_SELECT) OTE(DIE_CUSHION_2_PAD_R_SELECT) ,XIC(DIE_CUSHION_2_PAD_LEFT_SELECT) XIO(DIE_CUSHION_1_PAD_SELECT) XIO(DIE_CUSHION_2_PAD_SELECT) XIO(DIE_CUSHION_2_PAD_RIGHT_SELECT) OTE(DIE_CUSHION_2_PAD_L_SELECT) ];
   8: [XIC(DIE_CUSHION_1_PAD_SELECTED) ,XIC(DIE_CUSHION_2_PAD_SELECT_RL) ,XIC(DIE_CUSHION_2_PAD_R_SELECT) ]XIC(SAFETY_BAR_OPENED)XIC(MAIN_PRESS_CONDITION_DOWN)OTE(RIGHT_DIECUSHION_CONDITION);
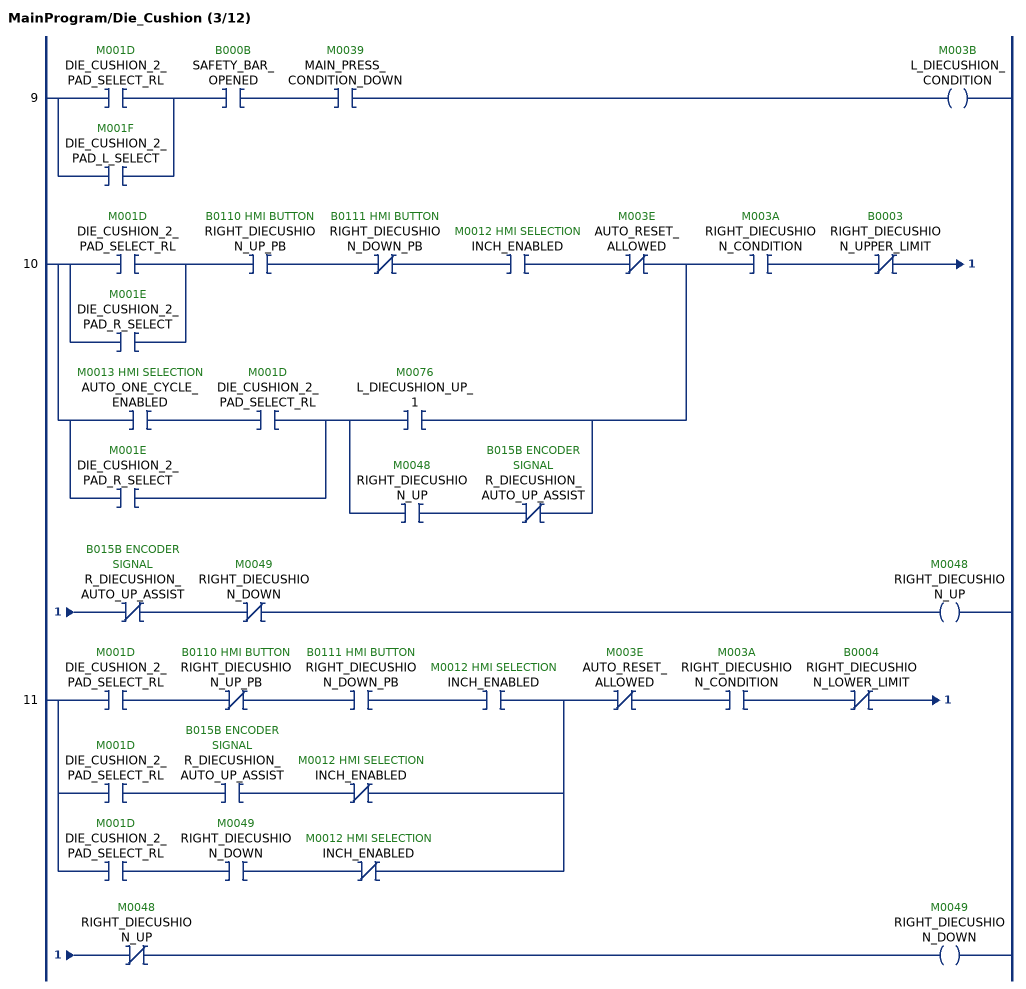
   9: [XIC(DIE_CUSHION_2_PAD_SELECT_RL) ,XIC(DIE_CUSHION_2_PAD_L_SELECT) ]XIC(SAFETY_BAR_OPENED)XIC(MAIN_PRESS_CONDITION_DOWN)OTE(L_DIECUSHION_CONDITION);
   10: [[XIC(DIE_CUSHION_2_PAD_SELECT_RL) ,XIC(DIE_CUSHION_2_PAD_R_SELECT) ] XIC(RIGHT_DIECUSHION_UP_PB) XIO(RIGHT_DIECUSHION_DOWN_PB) XIC(INCH_ENABLED) XIO(AUTO_RESET_ALLOWED) ,[XIC(AUTO_ONE_CYCLE_ENABLED) XIC(DIE_CUSHION_2_PAD_SELECT_RL) ,XIC(DIE_CUSHION_2_PAD_R_SELECT) ] [XIC(L_DIECUSHION_UP_1) ,XIC(RIGHT_DIECUSHION_UP) XIO(R_DIECUSHION_AUTO_UP_ASSIST) ] ]XIC(RIGHT_DIECUSHION_CONDITION)XIO(RIGHT_DIECUSHION_UPPER_LIMIT)XIO(R_DIECUSHION_AUTO_UP_ASSIST)XIO(RIGHT_DIECUSHION_DOWN)OTE(RIGHT_DIECUSHION_UP);
   11: [XIC(DIE_CUSHION_2_PAD_SELECT_RL) XIO(RIGHT_DIECUSHION_UP_PB) XIC(RIGHT_DIECUSHION_DOWN_PB) XIC(INCH_ENABLED) ,XIC(DIE_CUSHION_2_PAD_SELECT_RL) XIC(R_DIECUSHION_AUTO_UP_ASSIST) XIO(INCH_ENABLED) ,XIC(DIE_CUSHION_2_PAD_SELECT_RL) XIC(RIGHT_DIECUSHION_DOWN) XIO(INCH_ENABLED) ]XIO(AUTO_RESET_ALLOWED)XIC(RIGHT_DIECUSHION_CONDITION)XIO(RIGHT_DIECUSHION_LOWER_LIMIT)XIO(RIGHT_DIECUSHION_UP)OTE(RIGHT_DIECUSHION_DOWN);
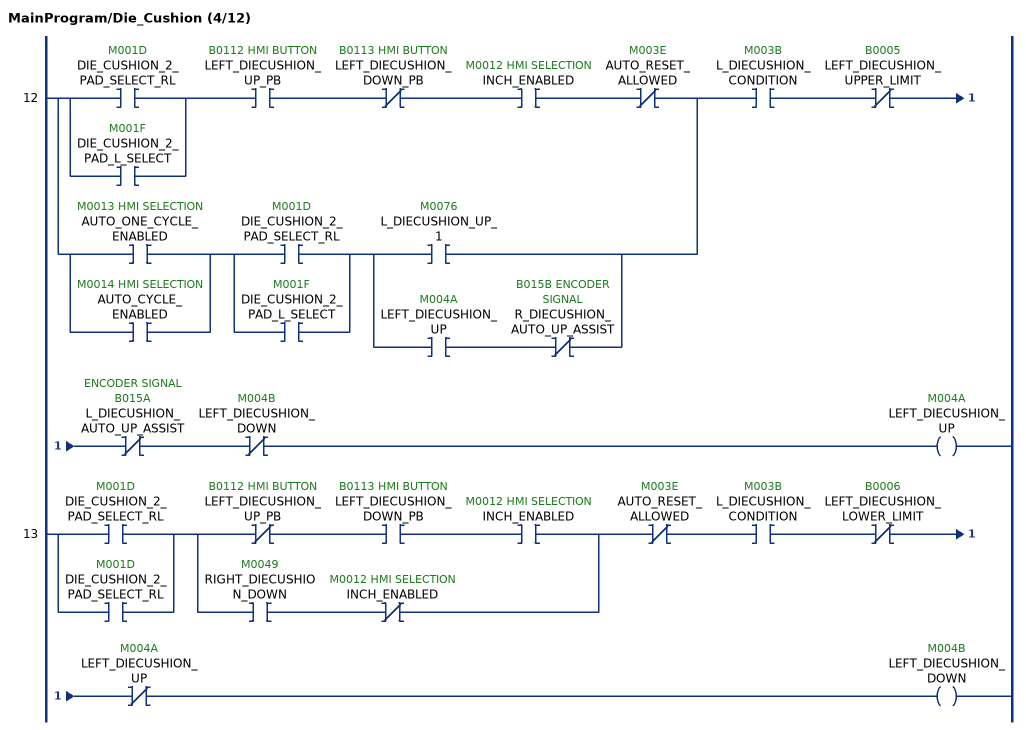
   12: [[XIC(DIE_CUSHION_2_PAD_SELECT_RL) ,XIC(DIE_CUSHION_2_PAD_L_SELECT) ] XIC(LEFT_DIECUSHION_UP_PB) XIO(LEFT_DIECUSHION_DOWN_PB) XIC(INCH_ENABLED) XIO(AUTO_RESET_ALLOWED) ,[XIC(AUTO_ONE_CYCLE_ENABLED) ,XIC(AUTO_CYCLE_ENABLED) ] [XIC(DIE_CUSHION_2_PAD_SELECT_RL) ,XIC(DIE_CUSHION_2_PAD_L_SELECT) ] [XIC(L_DIECUSHION_UP_1) ,XIC(LEFT_DIECUSHION_UP) XIO(R_DIECUSHION_AUTO_UP_ASSIST) ] ]XIC(L_DIECUSHION_CONDITION)XIO(LEFT_DIECUSHION_UPPER_LIMIT)XIO(L_DIECUSHION_AUTO_UP_ASSIST)XIO(LEFT_DIECUSHION_DOWN)OTE(LEFT_DIECUSHION_UP);
   13: [XIC(DIE_CUSHION_2_PAD_SELECT_RL) ,XIC(DIE_CUSHION_2_PAD_SELECT_RL) ][XIO(LEFT_DIECUSHION_UP_PB) XIC(LEFT_DIECUSHION_DOWN_PB) XIC(INCH_ENABLED) ,XIC(RIGHT_DIECUSHION_DOWN) XIO(INCH_ENABLED) ]XIO(AUTO_RESET_ALLOWED)XIC(L_DIECUSHION_CONDITION)XIO(LEFT_DIECUSHION_LOWER_LIMIT)XIO(LEFT_DIECUSHION_UP)OTE(LEFT_DIECUSHION_DOWN);
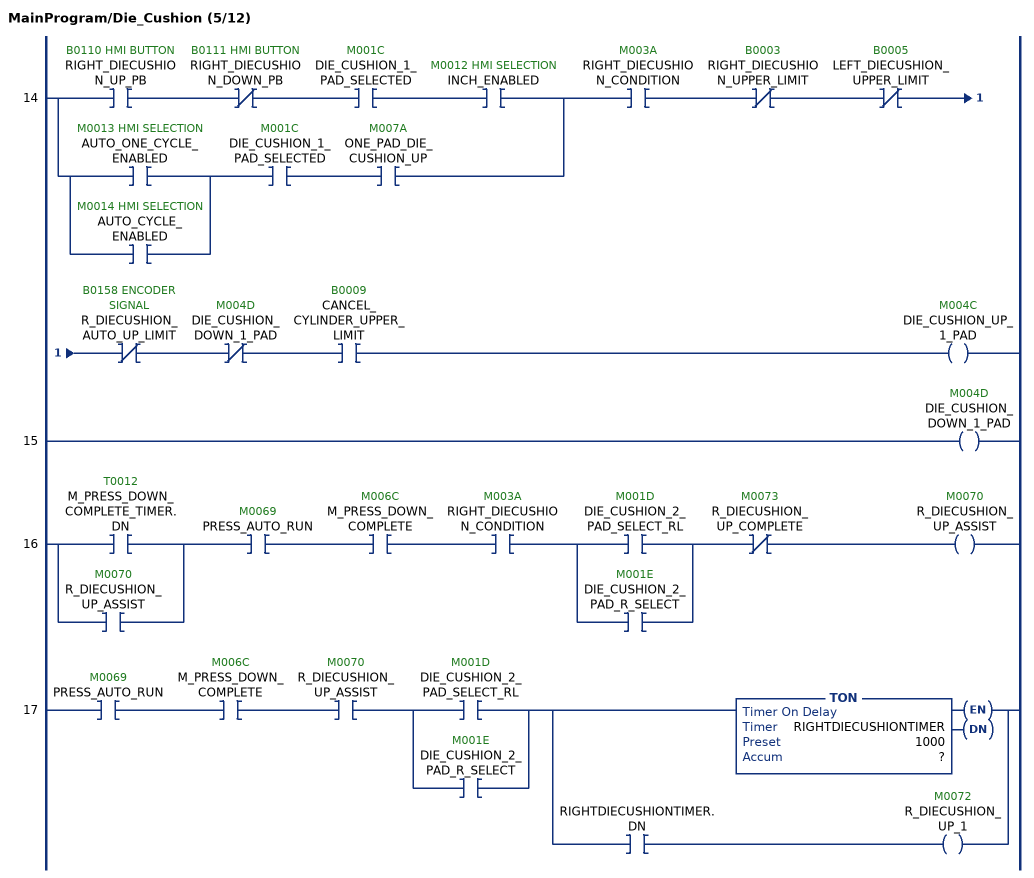
   14: [XIC(RIGHT_DIECUSHION_UP_PB) XIO(RIGHT_DIECUSHION_DOWN_PB) XIC(DIE_CUSHION_1_PAD_SELECTED) XIC(INCH_ENABLED) ,[XIC(AUTO_ONE_CYCLE_ENABLED) ,XIC(AUTO_CYCLE_ENABLED) ] XIC(DIE_CUSHION_1_PAD_SELECTED) XIC(ONE_PAD_DIE_CUSHION_UP) ]XIC(RIGHT_DIECUSHION_CONDITION)XIO(RIGHT_DIECUSHION_UPPER_LIMIT)XIO(LEFT_DIECUSHION_UPPER_LIMIT)XIO(R_DIECUSHION_AUTO_UP_LIMIT)XIO(DIE_CUSHION_DOWN_1_PAD)XIC(CANCEL_CYLINDER_UPPER_LIMIT)OTE(DIE_CUSHION_UP_1_PAD);
   15: OTE(DIE_CUSHION_DOWN_1_PAD);
   16: [XIC(M_PRESS_DOWN_COMPLETE_TIMER.DN) ,XIC(R_DIECUSHION_UP_ASSIST) ]XIC(PRESS_AUTO_RUN)XIC(M_PRESS_DOWN_COMPLETE)XIC(RIGHT_DIECUSHION_CONDITION)[XIC(DIE_CUSHION_2_PAD_SELECT_RL) ,XIC(DIE_CUSHION_2_PAD_R_SELECT) ]XIO(R_DIECUSHION_UP_COMPLETE)OTE(R_DIECUSHION_UP_ASSIST);
   17: XIC(PRESS_AUTO_RUN)XIC(M_PRESS_DOWN_COMPLETE)XIC(R_DIECUSHION_UP_ASSIST)[XIC(DIE_CUSHION_2_PAD_SELECT_RL) ,XIC(DIE_CUSHION_2_PAD_R_SELECT) ][TON(RIGHTDIECUSHIONTIMER,?,?) ,XIC(RIGHTDIECUSHIONTIMER.DN) OTE(R_DIECUSHION_UP_1) ];
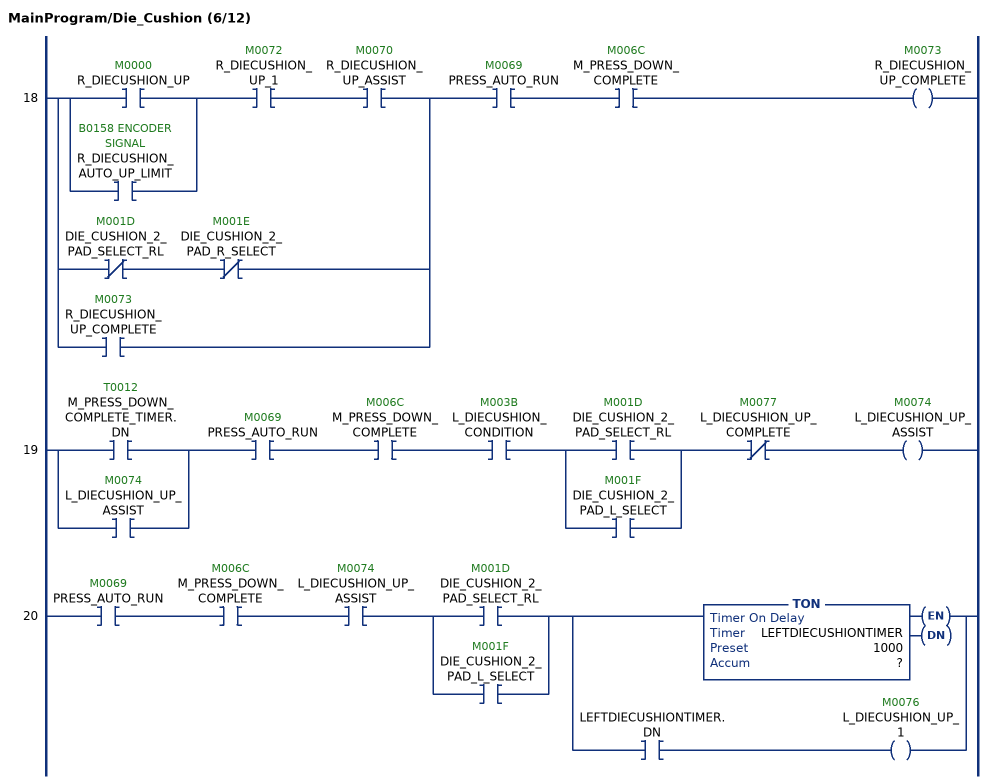
   18: [[XIC(R_DIECUSHION_UP) ,XIC(R_DIECUSHION_AUTO_UP_LIMIT) ] XIC(R_DIECUSHION_UP_1) XIC(R_DIECUSHION_UP_ASSIST) ,XIO(DIE_CUSHION_2_PAD_SELECT_RL) XIO(DIE_CUSHION_2_PAD_R_SELECT) ,XIC(R_DIECUSHION_UP_COMPLETE) ]XIC(PRESS_AUTO_RUN)XIC(M_PRESS_DOWN_COMPLETE)OTE(R_DIECUSHION_UP_COMPLETE);
   19: [XIC(M_PRESS_DOWN_COMPLETE_TIMER.DN) ,XIC(L_DIECUSHION_UP_ASSIST) ]XIC(PRESS_AUTO_RUN)XIC(M_PRESS_DOWN_COMPLETE)XIC(L_DIECUSHION_CONDITION)[XIC(DIE_CUSHION_2_PAD_SELECT_RL) ,XIC(DIE_CUSHION_2_PAD_L_SELECT) ]XIO(L_DIECUSHION_UP_COMPLETE)OTE(L_DIECUSHION_UP_ASSIST);
   20: XIC(PRESS_AUTO_RUN)XIC(M_PRESS_DOWN_COMPLETE)XIC(L_DIECUSHION_UP_ASSIST)[XIC(DIE_CUSHION_2_PAD_SELECT_RL) ,XIC(DIE_CUSHION_2_PAD_L_SELECT) ][TON(LEFTDIECUSHIONTIMER,?,?) ,XIC(LEFTDIECUSHIONTIMER.DN) OTE(L_DIECUSHION_UP_1) ];
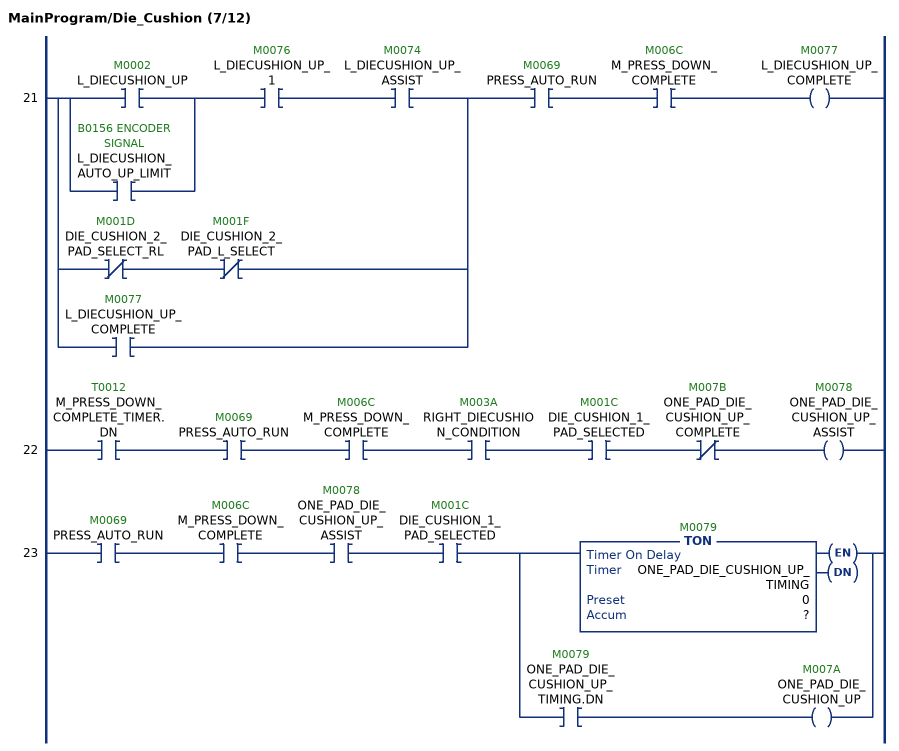
   21: [[XIC(L_DIECUSHION_UP) ,XIC(L_DIECUSHION_AUTO_UP_LIMIT) ] XIC(L_DIECUSHION_UP_1) XIC(L_DIECUSHION_UP_ASSIST) ,XIO(DIE_CUSHION_2_PAD_SELECT_RL) XIO(DIE_CUSHION_2_PAD_L_SELECT) ,XIC(L_DIECUSHION_UP_COMPLETE) ]XIC(PRESS_AUTO_RUN)XIC(M_PRESS_DOWN_COMPLETE)OTE(L_DIECUSHION_UP_COMPLETE);
   22: XIC(M_PRESS_DOWN_COMPLETE_TIMER.DN)XIC(PRESS_AUTO_RUN)XIC(M_PRESS_DOWN_COMPLETE)XIC(RIGHT_DIECUSHION_CONDITION)XIC(DIE_CUSHION_1_PAD_SELECTED)XIO(ONE_PAD_DIE_CUSHION_UP_COMPLETE)OTE(ONE_PAD_DIE_CUSHION_UP_ASSIST);
   23: XIC(PRESS_AUTO_RUN)XIC(M_PRESS_DOWN_COMPLETE)XIC(ONE_PAD_DIE_CUSHION_UP_ASSIST)XIC(DIE_CUSHION_1_PAD_SELECTED)[TON(ONE_PAD_DIE_CUSHION_UP_TIMING,?,?) ,XIC(ONE_PAD_DIE_CUSHION_UP_TIMING.DN) OTE(ONE_PAD_DIE_CUSHION_UP) ];
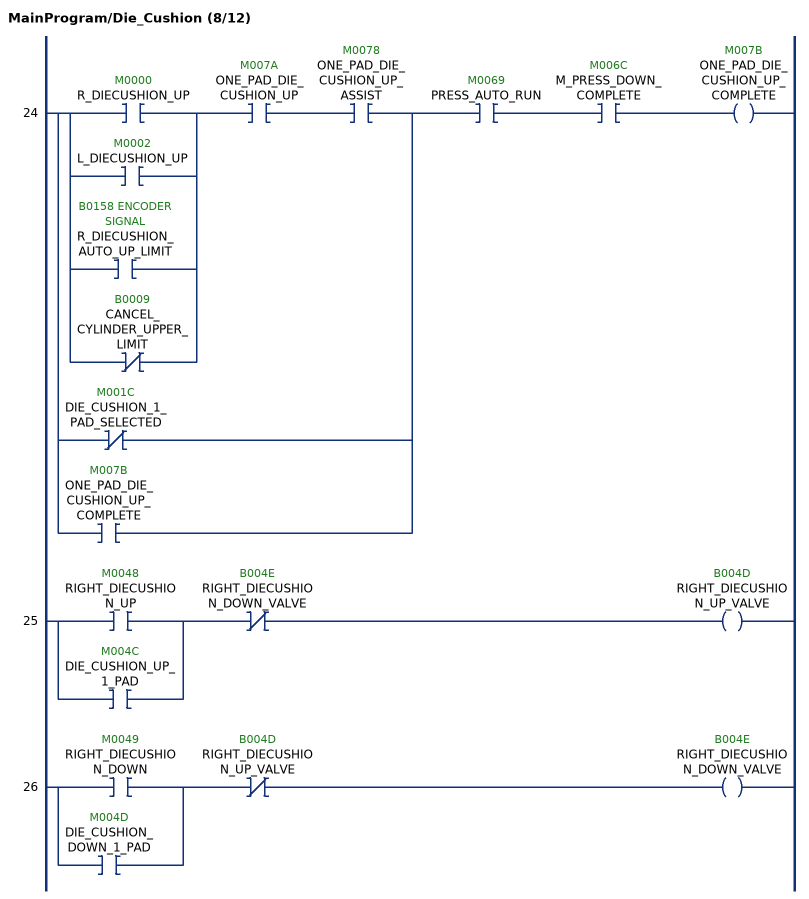
   24: [[XIC(R_DIECUSHION_UP) ,XIC(L_DIECUSHION_UP) ,XIC(R_DIECUSHION_AUTO_UP_LIMIT) ,XIO(CANCEL_CYLINDER_UPPER_LIMIT) ] XIC(ONE_PAD_DIE_CUSHION_UP) XIC(ONE_PAD_DIE_CUSHION_UP_ASSIST) ,XIO(DIE_CUSHION_1_PAD_SELECTED) ,XIC(ONE_PAD_DIE_CUSHION_UP_COMPLETE) ]XIC(PRESS_AUTO_RUN)XIC(M_PRESS_DOWN_COMPLETE)OTE(ONE_PAD_DIE_CUSHION_UP_COMPLETE);
   25: [XIC(RIGHT_DIECUSHION_UP) ,XIC(DIE_CUSHION_UP_1_PAD) ]XIO(RIGHT_DIECUSHION_DOWN_VALVE)OTE(RIGHT_DIECUSHION_UP_VALVE);
   26: [XIC(RIGHT_DIECUSHION_DOWN) ,XIC(DIE_CUSHION_DOWN_1_PAD) ]XIO(RIGHT_DIECUSHION_UP_VALVE)OTE(RIGHT_DIECUSHION_DOWN_VALVE);
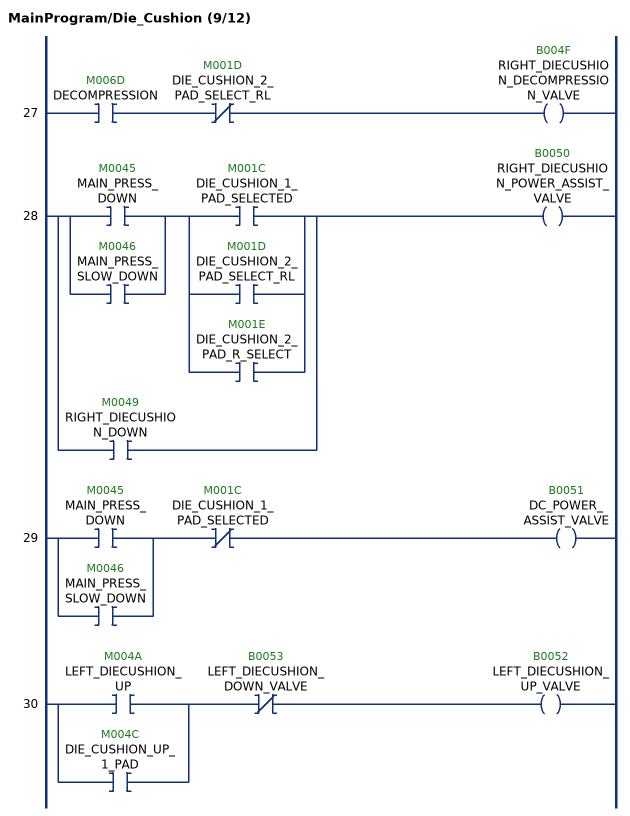
   27: XIC(DECOMPRESSION)XIO(DIE_CUSHION_2_PAD_SELECT_RL)OTE(RIGHT_DIECUSHION_DECOMPRESSION_VALVE);
   28: [[XIC(MAIN_PRESS_DOWN) ,XIC(MAIN_PRESS_SLOW_DOWN) ] [XIC(DIE_CUSHION_1_PAD_SELECTED) ,XIC(DIE_CUSHION_2_PAD_SELECT_RL) ,XIC(DIE_CUSHION_2_PAD_R_SELECT) ] ,XIC(RIGHT_DIECUSHION_DOWN) ]OTE(RIGHT_DIECUSHION_POWER_ASSIST_VALVE);
   29: [XIC(MAIN_PRESS_DOWN) ,XIC(MAIN_PRESS_SLOW_DOWN) ]XIO(DIE_CUSHION_1_PAD_SELECTED)OTE(DC_POWER_ASSIST_VALVE);
   30: [XIC(LEFT_DIECUSHION_UP) ,XIC(DIE_CUSHION_UP_1_PAD) ]XIO(LEFT_DIECUSHION_DOWN_VALVE)OTE(LEFT_DIECUSHION_UP_VALVE);
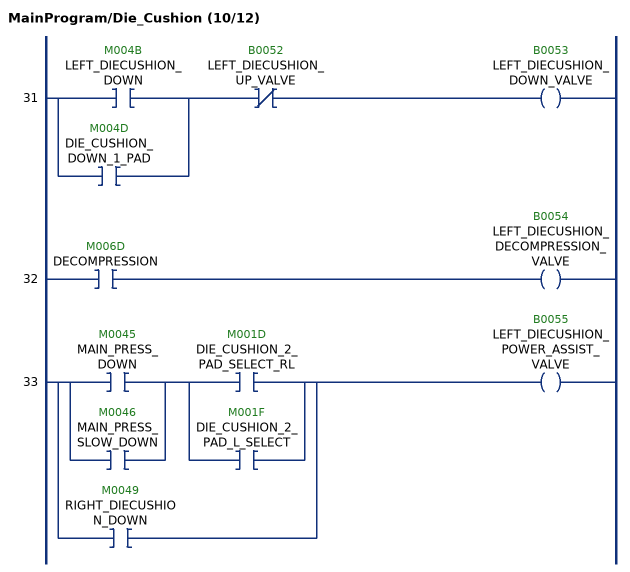
   31: [XIC(LEFT_DIECUSHION_DOWN) ,XIC(DIE_CUSHION_DOWN_1_PAD) ]XIO(LEFT_DIECUSHION_UP_VALVE)OTE(LEFT_DIECUSHION_DOWN_VALVE);
   32: XIC(DECOMPRESSION)OTE(LEFT_DIECUSHION_DECOMPRESSION_VALVE);
   33: [[XIC(MAIN_PRESS_DOWN) ,XIC(MAIN_PRESS_SLOW_DOWN) ] [XIC(DIE_CUSHION_2_PAD_SELECT_RL) ,XIC(DIE_CUSHION_2_PAD_L_SELECT) ] ,XIC(RIGHT_DIECUSHION_DOWN) ]OTE(LEFT_DIECUSHION_POWER_ASSIST_VALVE);
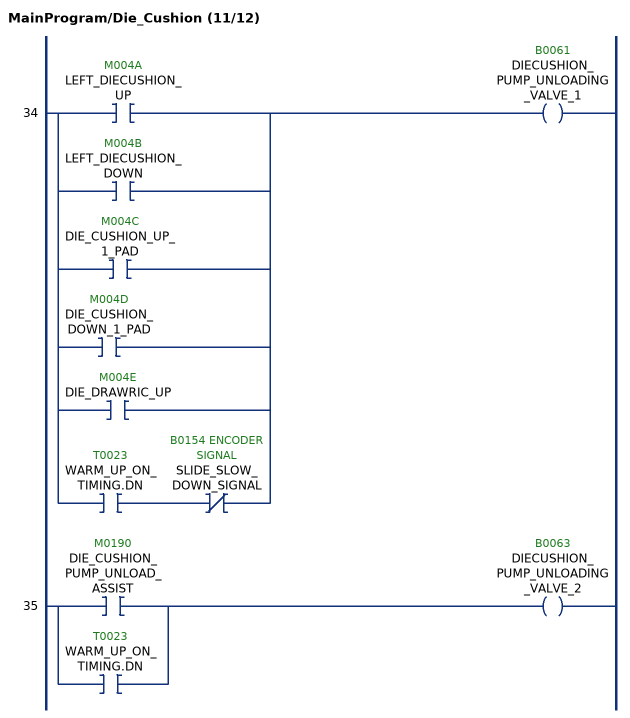
   34: [XIC(LEFT_DIECUSHION_UP) ,XIC(LEFT_DIECUSHION_DOWN) ,XIC(DIE_CUSHION_UP_1_PAD) ,XIC(DIE_CUSHION_DOWN_1_PAD) ,XIC(DIE_DRAWRIC_UP) ,XIC(WARM_UP_ON_TIMING.DN) XIO(SLIDE_SLOW_DOWN_SIGNAL) ]OTE(DIECUSHION_PUMP_UNLOADING_VALVE_1);
   35: [XIC(DIE_CUSHION_PUMP_UNLOAD_ASSIST) ,XIC(WARM_UP_ON_TIMING.DN) ]OTE(DIECUSHION_PUMP_UNLOADING_VALVE_2);
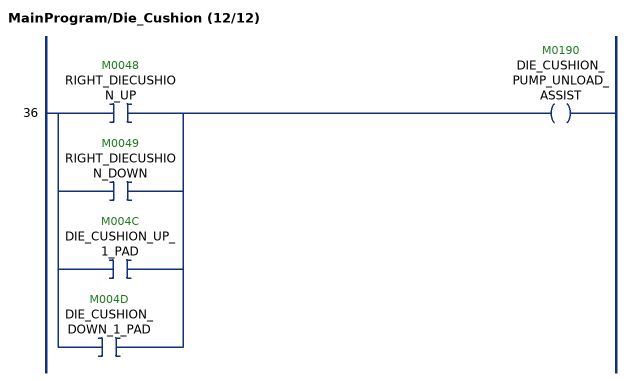
   36: [XIC(RIGHT_DIECUSHION_UP) ,XIC(RIGHT_DIECUSHION_DOWN) ,XIC(DIE_CUSHION_UP_1_PAD) ,XIC(DIE_CUSHION_DOWN_1_PAD) ]OTE(DIE_CUSHION_PUMP_UNLOAD_ASSIST);
END_ROUTINE
